   DATA[1580,22] := 1.713645;
   DATA[1580,23] := 795.0654;
   DATA[1580,24] := 2.0;
   DATA[1580,25] := 2.0;
   DATA[1580,26] := 7.876378;
   DATA[1580,27] := 142.8608;
   DATA[1580,28] := 262.8172;
   DATA[1580,29] := 12.11228;
   DATA[1580,30] := 1.724301;
   DATA[1580,31] := 1.291789;
   DATA[1580,32] := 0.7391096;
   DATA[1580,33] := 0.3081703;
   DATA[1580,34] := 2.0;
   DATA[1580,35] := 250.4166;
   DATA[1580,36] := 1.665972;
   DATA[1580,37] := 189.1182;
   DATA[1580,38] := 0.000128152;
   DATA[1580,39] := 1.0;
   DATA[1581,1] := 813.9059;
   DATA[1581,2] := 1.0;
   DATA[1581,3] := 1.0;
   DATA[1581,4] := 262.4968;
   DATA[1581,5] := 8.464369;
   DATA[1581,6] := 319.3027;
   DATA[1581,8] := 1.0;
   DATA[1581,9] := 1.0;
   DATA[1581,10] := 1.0;
   DATA[1581,11] := 19.70677;
   DATA[1581,12] := 2.214265;
   DATA[1581,13] := 907.7801;
   DATA[1581,14] := 1.0;
   DATA[1581,15] := 2.0;
   DATA[1581,16] := 1.0;
   DATA[1581,17] := 1.0;
   DATA[1581,18] := 1.0;
   DATA[1581,19] := 2.0;
   DATA[1581,20] := 148.808;
   DATA[1581,21] := 153.858;
   DATA[1581,22] := 1.713645;
   DATA[1581,23] := 795.2961;
   DATA[1581,24] := 2.0;
   DATA[1581,25] := 2.0;
   DATA[1581,26] := 7.876378;
   DATA[1581,27] := 142.8608;
   DATA[1581,28] := 262.8172;
   DATA[1581,29] := 12.11228;
   DATA[1581,30] := 1.725711;
   DATA[1581,31] := 1.291149;
   DATA[1581,32] := 0.736421;
   DATA[1581,33] := 0.3081703;
   DATA[1581,34] := 2.0;
   DATA[1581,35] := 250.4166;
   DATA[1581,36] := 1.665972;
   DATA[1581,37] := 189.2143;
   DATA[1581,38] := 0.000128152;
   DATA[1581,39] := 1.0;
   DATA[1582,1] := 813.7882;
   DATA[1582,2] := 1.0;
   DATA[1582,3] := 1.0;
   DATA[1582,4] := 262.4968;
   DATA[1582,5] := 8.464369;
   DATA[1582,6] := 319.2771;
   DATA[1582,8] := 1.0;
   DATA[1582,9] := 1.0;
   DATA[1582,10] := 1.0;
   DATA[1582,11] := 19.70677;
   DATA[1582,12] := 2.214265;
   DATA[1582,13] := 907.6199;
   DATA[1582,14] := 1.0;
   DATA[1582,15] := 2.0;
   DATA[1582,16] := 1.0;
   DATA[1582,17] := 1.0;
   DATA[1582,18] := 1.0;
   DATA[1582,19] := 2.0;
   DATA[1582,20] := 148.808;
   DATA[1582,21] := 153.858;
   DATA[1582,22] := 1.713645;
   DATA[1582,23] := 795.3345;
   DATA[1582,24] := 2.0;
   DATA[1582,25] := 2.0;
   DATA[1582,26] := 7.876378;
   DATA[1582,27] := 143.1684;
   DATA[1582,28] := 262.8172;
   DATA[1582,29] := 12.11228;
   DATA[1582,30] := 1.726609;
   DATA[1582,31] := 1.282439;
   DATA[1582,32] := 0.7346286;
   DATA[1582,33] := 0.306761;
   DATA[1582,34] := 2.0;
   DATA[1582,35] := 250.4166;
   DATA[1582,36] := 1.665972;
   DATA[1582,37] := 189.2143;
   DATA[1582,38] := 0.000128152;
   DATA[1582,39] := 1.0;
   DATA[1583,1] := 813.9059;
   DATA[1583,2] := 1.0;
   DATA[1583,3] := 1.0;
   DATA[1583,4] := 262.4968;
   DATA[1583,5] := 8.465651;
   DATA[1583,6] := 319.2258;
   DATA[1583,8] := 1.0;
   DATA[1583,9] := 1.0;
   DATA[1583,10] := 1.0;
   DATA[1583,11] := 19.70677;
   DATA[1583,12] := 2.214265;
   DATA[1583,13] := 906.8989;
   DATA[1583,14] := 1.0;
   DATA[1583,15] := 2.0;
   DATA[1583,16] := 1.0;
   DATA[1583,17] := 1.0;
   DATA[1583,18] := 1.0;
   DATA[1583,19] := 2.0;
   DATA[1583,20] := 148.808;
   DATA[1583,21] := 153.858;
   DATA[1583,22] := 1.715952;
   DATA[1583,23] := 795.7575;
   DATA[1583,24] := 2.0;
   DATA[1583,25] := 2.0;
   DATA[1583,26] := 7.876378;
   DATA[1583,27] := 143.1684;
   DATA[1583,28] := 262.8172;
   DATA[1583,29] := 12.11228;
   DATA[1583,30] := 1.726609;
   DATA[1583,31] := 1.269502;
   DATA[1583,32] := 0.7346286;
   DATA[1583,33] := 0.306761;
   DATA[1583,34] := 2.0;
   DATA[1583,35] := 250.4166;
   DATA[1583,36] := 1.665972;
   DATA[1583,37] := 189.2143;
   DATA[1583,38] := 0.000128152;
   DATA[1583,39] := 1.0;
   DATA[1584,1] := 813.6312;
   DATA[1584,2] := 1.0;
   DATA[1584,3] := 1.0;
   DATA[1584,4] := 262.4968;
   DATA[1584,5] := 8.465651;
   DATA[1584,6] := 319.072;
   DATA[1584,8] := 1.0;
   DATA[1584,9] := 1.0;
   DATA[1584,10] := 1.0;
   DATA[1584,11] := 19.67155;
   DATA[1584,12] := 2.214265;
   DATA[1584,13] := 906.4583;
   DATA[1584,14] := 1.0;
   DATA[1584,15] := 2.0;
   DATA[1584,16] := 1.0;
   DATA[1584,17] := 1.0;
   DATA[1584,18] := 1.0;
   DATA[1584,19] := 2.0;
   DATA[1584,20] := 148.808;
   DATA[1584,21] := 153.858;
   DATA[1584,22] := 1.715952;
   DATA[1584,23] := 795.6806;
   DATA[1584,24] := 2.0;
   DATA[1584,25] := 2.0;
   DATA[1584,26] := 7.876378;
   DATA[1584,27] := 143.1684;
   DATA[1584,28] := 262.8172;
   DATA[1584,29] := 12.11228;
   DATA[1584,30] := 1.726609;
   DATA[1584,31] := 1.261304;
   DATA[1584,32] := 0.7346286;
   DATA[1584,33] := 0.306761;
   DATA[1584,34] := 2.0;
   DATA[1584,35] := 250.4166;
   DATA[1584,36] := 1.665972;
   DATA[1584,37] := 189.2143;
   DATA[1584,38] := 0.000128152;
   DATA[1584,39] := 1.0;
   DATA[1585,1] := 813.5919;
   DATA[1585,2] := 1.0;
   DATA[1585,3] := 1.0;
   DATA[1585,4] := 262.6891;
   DATA[1585,5] := 8.465651;
   DATA[1585,6] := 319.072;
   DATA[1585,8] := 1.0;
   DATA[1585,9] := 1.0;
   DATA[1585,10] := 1.0;
   DATA[1585,11] := 19.67155;
   DATA[1585,12] := 2.214265;
   DATA[1585,13] := 905.6172;
   DATA[1585,14] := 1.0;
   DATA[1585,15] := 2.0;
   DATA[1585,16] := 1.0;
   DATA[1585,17] := 1.0;
   DATA[1585,18] := 1.0;
   DATA[1585,19] := 2.0;
   DATA[1585,20] := 148.808;
   DATA[1585,21] := 153.858;
   DATA[1585,22] := 1.713389;
   DATA[1585,23] := 795.796;
   DATA[1585,24] := 2.0;
   DATA[1585,25] := 2.0;
   DATA[1585,26] := 7.876378;
   DATA[1585,27] := 143.1684;
   DATA[1585,28] := 262.8172;
   DATA[1585,29] := 12.11228;
   DATA[1585,30] := 1.726609;
   DATA[1585,31] := 1.26361;
   DATA[1585,32] := 0.7346286;
   DATA[1585,33] := 0.3084265;
   DATA[1585,34] := 2.0;
   DATA[1585,35] := 250.4166;
   DATA[1585,36] := 1.665972;
   DATA[1585,37] := 189.2143;
   DATA[1585,38] := 0.000128152;
   DATA[1585,39] := 1.0;
   DATA[1586,1] := 813.3956;
   DATA[1586,2] := 1.0;
   DATA[1586,3] := 1.0;
   DATA[1586,4] := 262.6891;
   DATA[1586,5] := 8.465651;
   DATA[1586,6] := 319.072;
   DATA[1586,8] := 1.0;
   DATA[1586,9] := 1.0;
   DATA[1586,10] := 1.0;
   DATA[1586,11] := 19.67155;
   DATA[1586,12] := 2.212856;
   DATA[1586,13] := 905.7774;
   DATA[1586,14] := 1.0;
   DATA[1586,15] := 2.0;
   DATA[1586,16] := 1.0;
   DATA[1586,17] := 1.0;
   DATA[1586,18] := 1.0;
   DATA[1586,19] := 2.0;
   DATA[1586,20] := 148.808;
   DATA[1586,21] := 153.858;
   DATA[1586,22] := 1.713004;
   DATA[1586,23] := 795.796;
   DATA[1586,24] := 2.0;
   DATA[1586,25] := 2.0;
   DATA[1586,26] := 7.874776;
   DATA[1586,27] := 143.0659;
   DATA[1586,28] := 262.8172;
   DATA[1586,29] := 12.11228;
   DATA[1586,30] := 1.726865;
   DATA[1586,31] := 1.271039;
   DATA[1586,32] := 0.7357808;
   DATA[1586,33] := 0.3084265;
   DATA[1586,34] := 2.0;
   DATA[1586,35] := 250.4166;
   DATA[1586,36] := 1.665972;
   DATA[1586,37] := 189.2143;
   DATA[1586,38] := 0.000128152;
   DATA[1586,39] := 1.0;
   DATA[1587,1] := 814.0237;
   DATA[1587,2] := 1.0;
   DATA[1587,3] := 1.0;
   DATA[1587,4] := 262.6891;
   DATA[1587,5] := 8.465651;
   DATA[1587,6] := 319.072;
   DATA[1587,8] := 1.0;
   DATA[1587,9] := 1.0;
   DATA[1587,10] := 1.0;
   DATA[1587,11] := 19.71637;
   DATA[1587,12] := 2.2126;
   DATA[1587,13] := 904.9763;
   DATA[1587,14] := 1.0;
   DATA[1587,15] := 2.0;
   DATA[1587,16] := 1.0;
   DATA[1587,17] := 1.0;
   DATA[1587,18] := 1.0;
   DATA[1587,19] := 2.0;
   DATA[1587,20] := 148.808;
   DATA[1587,21] := 153.9862;
   DATA[1587,22] := 1.713004;
   DATA[1587,23] := 796.1036;
   DATA[1587,24] := 2.0;
   DATA[1587,25] := 2.0;
   DATA[1587,26] := 7.874776;
   DATA[1587,27] := 143.0659;
   DATA[1587,28] := 262.8172;
   DATA[1587,29] := 12.11228;
   DATA[1587,30] := 1.726865;
   DATA[1587,31] := 1.280902;
   DATA[1587,32] := 0.7357808;
   DATA[1587,33] := 0.3084265;
   DATA[1587,34] := 2.0;
   DATA[1587,35] := 250.4166;
   DATA[1587,36] := 1.665972;
   DATA[1587,37] := 189.2143;
   DATA[1587,38] := 0.000128152;
   DATA[1587,39] := 1.0;
   DATA[1588,1] := 813.9844;
   DATA[1588,2] := 1.0;
   DATA[1588,3] := 1.0;
   DATA[1588,4] := 262.6891;
   DATA[1588,5] := 8.465651;
   DATA[1588,6] := 319.072;
   DATA[1588,8] := 1.0;
   DATA[1588,9] := 1.0;
   DATA[1588,10] := 1.0;
   DATA[1588,11] := 19.71637;
   DATA[1588,12] := 2.2126;
   DATA[1588,13] := 904.4957;
   DATA[1588,14] := 1.0;
   DATA[1588,15] := 2.0;
   DATA[1588,16] := 1.0;
   DATA[1588,17] := 1.0;
   DATA[1588,18] := 1.0;
   DATA[1588,19] := 2.0;
   DATA[1588,20] := 148.808;
   DATA[1588,21] := 153.9862;
   DATA[1588,22] := 1.713004;
   DATA[1588,23] := 796.1805;
   DATA[1588,24] := 2.0;
   DATA[1588,25] := 2.0;
   DATA[1588,26] := 7.874776;
   DATA[1588,27] := 143.0659;
   DATA[1588,28] := 262.8172;
   DATA[1588,29] := 12.11228;
   DATA[1588,30] := 1.726865;
   DATA[1588,31] := 1.28167;
   DATA[1588,32] := 0.7357808;
   DATA[1588,33] := 0.3084265;
   DATA[1588,34] := 2.0;
   DATA[1588,35] := 250.4166;
   DATA[1588,36] := 1.665972;
   DATA[1588,37] := 189.2143;
   DATA[1588,38] := 0.000128152;
   DATA[1588,39] := 1.0;
   DATA[1589,1] := 813.7489;
   DATA[1589,2] := 1.0;
   DATA[1589,3] := 1.0;
   DATA[1589,4] := 262.6891;
   DATA[1589,5] := 8.465651;
   DATA[1589,6] := 319.072;
   DATA[1589,8] := 1.0;
   DATA[1589,9] := 1.0;
   DATA[1589,10] := 1.0;
   DATA[1589,11] := 19.74838;
   DATA[1589,12] := 2.2126;
   DATA[1589,13] := 903.8948;
   DATA[1589,14] := 1.0;
   DATA[1589,15] := 2.0;
   DATA[1589,16] := 1.0;
   DATA[1589,17] := 1.0;
   DATA[1589,18] := 1.0;
   DATA[1589,19] := 2.0;
   DATA[1589,20] := 148.808;
   DATA[1589,21] := 153.9862;
   DATA[1589,22] := 1.71262;
   DATA[1589,23] := 795.9498;
   DATA[1589,24] := 2.0;
   DATA[1589,25] := 2.0;
   DATA[1589,26] := 7.874776;
   DATA[1589,27] := 143.0659;
   DATA[1589,28] := 262.8172;
   DATA[1589,29] := 12.11228;
   DATA[1589,30] := 1.726865;
   DATA[1589,31] := 1.279877;
   DATA[1589,32] := 0.7357808;
   DATA[1589,33] := 0.3084265;
   DATA[1589,34] := 2.0;
   DATA[1589,35] := 250.4166;
   DATA[1589,36] := 1.665972;
   DATA[1589,37] := 189.2143;
   DATA[1589,38] := 0.000128152;
   DATA[1589,39] := 1.0;
   DATA[1590,1] := 813.7489;
   DATA[1590,2] := 1.0;
   DATA[1590,3] := 1.0;
   DATA[1590,4] := 262.6891;
   DATA[1590,5] := 8.465651;
   DATA[1590,6] := 319.072;
   DATA[1590,8] := 1.0;
   DATA[1590,9] := 1.0;
   DATA[1590,10] := 1.0;
   DATA[1590,11] := 19.77079;
   DATA[1590,12] := 2.2126;
   DATA[1590,13] := 903.2941;
   DATA[1590,14] := 1.0;
   DATA[1590,15] := 2.0;
   DATA[1590,16] := 1.0;
   DATA[1590,17] := 1.0;
   DATA[1590,18] := 1.0;
   DATA[1590,19] := 2.0;
   DATA[1590,20] := 148.808;
   DATA[1590,21] := 153.9862;
   DATA[1590,22] := 1.711595;
   DATA[1590,23] := 796.3727;
   DATA[1590,24] := 2.0;
   DATA[1590,25] := 2.0;
   DATA[1590,26] := 7.874776;
   DATA[1590,27] := 143.0403;
   DATA[1590,28] := 262.8172;
   DATA[1590,29] := 11.92002;
   DATA[1590,30] := 1.726865;
   DATA[1590,31] := 1.279237;
   DATA[1590,32] := 0.7357808;
   DATA[1590,33] := 0.3084265;
   DATA[1590,34] := 2.0;
   DATA[1590,35] := 250.4166;
   DATA[1590,36] := 1.665972;
   DATA[1590,37] := 189.2143;
   DATA[1590,38] := 0.000128152;
   DATA[1590,39] := 1.0;
   DATA[1591,1] := 813.8275;
   DATA[1591,2] := 1.0;
   DATA[1591,3] := 1.0;
   DATA[1591,4] := 262.6891;
   DATA[1591,5] := 8.465651;
   DATA[1591,6] := 319.072;
   DATA[1591,8] := 1.0;
   DATA[1591,9] := 1.0;
   DATA[1591,10] := 1.0;
   DATA[1591,11] := 19.7996;
   DATA[1591,12] := 2.2126;
   DATA[1591,13] := 902.6532;
   DATA[1591,14] := 1.0;
   DATA[1591,15] := 2.0;
   DATA[1591,16] := 1.0;
   DATA[1591,17] := 1.0;
   DATA[1591,18] := 1.0;
   DATA[1591,19] := 2.0;
   DATA[1591,20] := 148.808;
   DATA[1591,21] := 153.9862;
   DATA[1591,22] := 1.711082;
   DATA[1591,23] := 796.5266;
   DATA[1591,24] := 2.0;
   DATA[1591,25] := 2.0;
   DATA[1591,26] := 7.874776;
   DATA[1591,27] := 143.0403;
   DATA[1591,28] := 262.8172;
   DATA[1591,29] := 11.92002;
   DATA[1591,30] := 1.726865;
   DATA[1591,31] := 1.28167;
   DATA[1591,32] := 0.7352687;
   DATA[1591,33] := 0.3084265;
   DATA[1591,34] := 2.0;
   DATA[1591,35] := 250.4166;
   DATA[1591,36] := 1.665972;
   DATA[1591,37] := 189.2143;
   DATA[1591,38] := 0.000128152;
   DATA[1591,39] := 1.0;
   DATA[1592,1] := 813.5134;
   DATA[1592,2] := 1.0;
   DATA[1592,3] := 1.0;
   DATA[1592,4] := 262.6891;
   DATA[1592,5] := 8.465651;
   DATA[1592,6] := 319.072;
   DATA[1592,8] := 1.0;
   DATA[1592,9] := 1.0;
   DATA[1592,10] := 1.0;
   DATA[1592,11] := 19.7996;
   DATA[1592,12] := 2.211318;
   DATA[1592,13] := 902.2126;
   DATA[1592,14] := 1.0;
   DATA[1592,15] := 2.0;
   DATA[1592,16] := 1.0;
   DATA[1592,17] := 1.0;
   DATA[1592,18] := 1.0;
   DATA[1592,19] := 2.0;
   DATA[1592,20] := 148.808;
   DATA[1592,21] := 153.9862;
   DATA[1592,22] := 1.7098;
   DATA[1592,23] := 796.4496;
   DATA[1592,24] := 2.0;
   DATA[1592,25] := 2.0;
   DATA[1592,26] := 7.874776;
   DATA[1592,27] := 143.0403;
   DATA[1592,28] := 262.8172;
   DATA[1592,29] := 11.92002;
   DATA[1592,30] := 1.726865;
   DATA[1592,31] := 1.291405;
   DATA[1592,32] := 0.7351407;
   DATA[1592,33] := 0.3084265;
   DATA[1592,34] := 2.0;
   DATA[1592,35] := 250.4166;
   DATA[1592,36] := 1.665972;
   DATA[1592,37] := 189.2143;
   DATA[1592,38] := 0.000128152;
   DATA[1592,39] := 1.0;
   DATA[1593,1] := 813.7489;
   DATA[1593,2] := 1.0;
   DATA[1593,3] := 1.0;
   DATA[1593,4] := 262.6891;
   DATA[1593,5] := 8.465651;
   DATA[1593,6] := 319.072;
   DATA[1593,8] := 1.0;
   DATA[1593,9] := 1.0;
   DATA[1593,10] := 1.0;
   DATA[1593,11] := 19.73878;
   DATA[1593,12] := 2.211318;
   DATA[1593,13] := 901.772;
   DATA[1593,14] := 1.0;
   DATA[1593,15] := 2.0;
   DATA[1593,16] := 1.0;
   DATA[1593,17] := 1.0;
   DATA[1593,18] := 1.0;
   DATA[1593,19] := 2.0;
   DATA[1593,20] := 148.808;
   DATA[1593,21] := 153.9862;
   DATA[1593,22] := 1.7098;
   DATA[1593,23] := 796.565;
   DATA[1593,24] := 2.0;
   DATA[1593,25] := 2.0;
   DATA[1593,26] := 7.874776;
   DATA[1593,27] := 143.0403;
   DATA[1593,28] := 262.8172;
   DATA[1593,29] := 11.92002;
   DATA[1593,30] := 1.726865;
   DATA[1593,31] := 1.285641;
   DATA[1593,32] := 0.7351407;
   DATA[1593,33] := 0.3084265;
   DATA[1593,34] := 2.0;
   DATA[1593,35] := 250.4166;
   DATA[1593,36] := 1.665972;
   DATA[1593,37] := 189.2143;
   DATA[1593,38] := 0.000128152;
   DATA[1593,39] := 1.0;
   DATA[1594,1] := 813.5919;
   DATA[1594,2] := 1.0;
   DATA[1594,3] := 1.0;
   DATA[1594,4] := 262.6891;
   DATA[1594,5] := 8.465651;
   DATA[1594,6] := 319.072;
   DATA[1594,8] := 1.0;
   DATA[1594,9] := 1.0;
   DATA[1594,10] := 1.0;
   DATA[1594,11] := 19.73878;
   DATA[1594,12] := 2.2126;
   DATA[1594,13] := 901.2914;
   DATA[1594,14] := 1.0;
   DATA[1594,15] := 2.0;
   DATA[1594,16] := 1.0;
   DATA[1594,17] := 1.0;
   DATA[1594,18] := 1.0;
   DATA[1594,19] := 2.0;
   DATA[1594,20] := 148.808;
   DATA[1594,21] := 153.9862;
   DATA[1594,22] := 1.7098;
   DATA[1594,23] := 797.1418;
   DATA[1594,24] := 2.0;
   DATA[1594,25] := 2.0;
   DATA[1594,26] := 7.874776;
   DATA[1594,27] := 142.8352;
   DATA[1594,28] := 262.8172;
   DATA[1594,29] := 11.92002;
   DATA[1594,30] := 1.726865;
   DATA[1594,31] := 1.289228;
   DATA[1594,32] := 0.7351407;
   DATA[1594,33] := 0.3084265;
   DATA[1594,34] := 2.0;
   DATA[1594,35] := 250.3044;
   DATA[1594,36] := 1.665972;
   DATA[1594,37] := 189.2143;
   DATA[1594,38] := 0.000128152;
   DATA[1594,39] := 1.0;
   DATA[1595,1] := 813.7882;
   DATA[1595,2] := 1.0;
   DATA[1595,3] := 1.0;
   DATA[1595,4] := 262.6891;
   DATA[1595,5] := 8.465651;
   DATA[1595,6] := 319.072;
   DATA[1595,8] := 1.0;
   DATA[1595,9] := 1.0;
   DATA[1595,10] := 1.0;
   DATA[1595,11] := 19.73878;
   DATA[1595,12] := 2.212856;
   DATA[1595,13] := 900.6906;
   DATA[1595,14] := 1.0;
   DATA[1595,15] := 2.0;
   DATA[1595,16] := 1.0;
   DATA[1595,17] := 1.0;
   DATA[1595,18] := 1.0;
   DATA[1595,19] := 2.0;
   DATA[1595,20] := 148.808;
   DATA[1595,21] := 153.9862;
   DATA[1595,22] := 1.7098;
   DATA[1595,23] := 797.0649;
   DATA[1595,24] := 2.0;
   DATA[1595,25] := 2.0;
   DATA[1595,26] := 7.877339;
   DATA[1595,27] := 142.8352;
   DATA[1595,28] := 262.8172;
   DATA[1595,29] := 11.92002;
   DATA[1595,30] := 1.726865;
   DATA[1595,31] := 1.291789;
   DATA[1595,32] := 0.7351407;
   DATA[1595,33] := 0.3084265;
   DATA[1595,34] := 2.0;
   DATA[1595,35] := 250.2724;
   DATA[1595,36] := 1.665972;
   DATA[1595,37] := 188.8939;
   DATA[1595,38] := 0.000128152;
   DATA[1595,39] := 1.0;
   DATA[1596,1] := 813.7882;
   DATA[1596,2] := 1.0;
   DATA[1596,3] := 1.0;
   DATA[1596,4] := 262.6891;
   DATA[1596,5] := 8.465651;
   DATA[1596,6] := 319.072;
   DATA[1596,8] := 1.0;
   DATA[1596,9] := 1.0;
   DATA[1596,10] := 1.0;
   DATA[1596,11] := 19.73878;
   DATA[1596,12] := 2.212856;
   DATA[1596,13] := 900.2499;
   DATA[1596,14] := 1.0;
   DATA[1596,15] := 2.0;
   DATA[1596,16] := 1.0;
   DATA[1596,17] := 1.0;
   DATA[1596,18] := 1.0;
   DATA[1596,19] := 2.0;
   DATA[1596,20] := 148.808;
   DATA[1596,21] := 153.9862;
   DATA[1596,22] := 1.7098;
   DATA[1596,23] := 797.2187;
   DATA[1596,24] := 2.0;
   DATA[1596,25] := 2.0;
   DATA[1596,26] := 7.877339;
   DATA[1596,27] := 142.8352;
   DATA[1596,28] := 262.8172;
   DATA[1596,29] := 12.26609;
   DATA[1596,30] := 1.725968;
   DATA[1596,31] := 1.291789;
   DATA[1596,32] := 0.7351407;
   DATA[1596,33] := 0.3084265;
   DATA[1596,34] := 2.0;
   DATA[1596,35] := 250.0801;
   DATA[1596,36] := 1.665972;
   DATA[1596,37] := 188.8779;
   DATA[1596,38] := 0.000128152;
   DATA[1596,39] := 1.0;
   DATA[1597,1] := 813.6312;
   DATA[1597,2] := 1.0;
   DATA[1597,3] := 1.0;
   DATA[1597,4] := 262.4648;
   DATA[1597,5] := 8.465651;
   DATA[1597,6] := 319.072;
   DATA[1597,8] := 1.0;
   DATA[1597,9] := 1.0;
   DATA[1597,10] := 1.0;
   DATA[1597,11] := 19.75159;
   DATA[1597,12] := 2.212856;
   DATA[1597,13] := 899.7693;
   DATA[1597,14] := 1.0;
   DATA[1597,15] := 2.0;
   DATA[1597,16] := 1.0;
   DATA[1597,17] := 1.0;
   DATA[1597,18] := 1.0;
   DATA[1597,19] := 2.0;
   DATA[1597,20] := 148.808;
   DATA[1597,21] := 153.9862;
   DATA[1597,22] := 1.7098;
   DATA[1597,23] := 797.4494;
   DATA[1597,24] := 2.0;
   DATA[1597,25] := 2.0;
   DATA[1597,26] := 7.877339;
   DATA[1597,27] := 142.8352;
   DATA[1597,28] := 262.8172;
   DATA[1597,29] := 12.26609;
   DATA[1597,30] := 1.724301;
   DATA[1597,31] := 1.301652;
   DATA[1597,32] := 0.7351407;
   DATA[1597,33] := 0.3084265;
   DATA[1597,34] := 2.0;
   DATA[1597,35] := 250.0801;
   DATA[1597,36] := 1.665972;
   DATA[1597,37] := 188.8779;
   DATA[1597,38] := 0.000128152;
   DATA[1597,39] := 1.0;
   DATA[1598,1] := 813.5134;
   DATA[1598,2] := 1.0;
   DATA[1598,3] := 1.0;
   DATA[1598,4] := 262.4648;
   DATA[1598,5] := 8.466612;
   DATA[1598,6] := 319.072;
   DATA[1598,8] := 1.0;
   DATA[1598,9] := 1.0;
   DATA[1598,10] := 1.0;
   DATA[1598,11] := 19.7804;
   DATA[1598,12] := 2.212856;
   DATA[1598,13] := 899.4489;
   DATA[1598,14] := 1.0;
   DATA[1598,15] := 2.0;
   DATA[1598,16] := 1.0;
   DATA[1598,17] := 1.0;
   DATA[1598,18] := 1.0;
   DATA[1598,19] := 2.0;
   DATA[1598,20] := 148.808;
   DATA[1598,21] := 153.9862;
   DATA[1598,22] := 1.7098;
   DATA[1598,23] := 797.5262;
   DATA[1598,24] := 2.0;
   DATA[1598,25] := 2.0;
   DATA[1598,26] := 7.877339;
   DATA[1598,27] := 143.0403;
   DATA[1598,28] := 262.8172;
   DATA[1598,29] := 12.26609;
   DATA[1598,30] := 1.722379;
   DATA[1598,31] := 1.294095;
   DATA[1598,32] := 0.7351407;
   DATA[1598,33] := 0.3074656;
   DATA[1598,34] := 2.0;
   DATA[1598,35] := 249.9359;
   DATA[1598,36] := 1.665972;
   DATA[1598,37] := 188.8779;
   DATA[1598,38] := 0.000128152;
   DATA[1598,39] := 1.0;
   DATA[1599,1] := 813.9059;
   DATA[1599,2] := 1.0;
   DATA[1599,3] := 1.0;
   DATA[1599,4] := 262.4648;
   DATA[1599,5] := 8.467573;
   DATA[1599,6] := 319.072;
   DATA[1599,8] := 1.0;
   DATA[1599,9] := 1.0;
   DATA[1599,10] := 1.0;
   DATA[1599,11] := 19.7964;
   DATA[1599,12] := 2.212856;
   DATA[1599,13] := 898.9282;
   DATA[1599,14] := 1.0;
   DATA[1599,15] := 2.0;
   DATA[1599,16] := 1.0;
   DATA[1599,17] := 1.0;
   DATA[1599,18] := 1.0;
   DATA[1599,19] := 2.0;
   DATA[1599,20] := 148.808;
   DATA[1599,21] := 153.9093;
   DATA[1599,22] := 1.7098;
   DATA[1599,23] := 797.4879;
   DATA[1599,24] := 2.0;
   DATA[1599,25] := 2.0;
   DATA[1599,26] := 7.877339;
   DATA[1599,27] := 143.0403;
   DATA[1599,28] := 262.8172;
   DATA[1599,29] := 12.26609;
   DATA[1599,30] := 1.722379;
   DATA[1599,31] := 1.291533;
   DATA[1599,32] := 0.7351407;
   DATA[1599,33] := 0.3074656;
   DATA[1599,34] := 2.0;
   DATA[1599,35] := 249.9359;
   DATA[1599,36] := 1.665972;
   DATA[1599,37] := 188.8779;
   DATA[1599,38] := 0.000128152;
   DATA[1599,39] := 1.0;
   DATA[1600,1] := 814.2985;
   DATA[1600,2] := 1.0;
   DATA[1600,3] := 1.0;
   DATA[1600,4] := 262.4648;
   DATA[1600,5] := 8.467573;
   DATA[1600,6] := 319.072;
   DATA[1600,8] := 1.0;
   DATA[1600,9] := 1.0;
   DATA[1600,10] := 1.0;
   DATA[1600,11] := 19.7964;
   DATA[1600,12] := 2.212856;
   DATA[1600,13] := 898.8481;
   DATA[1600,14] := 1.0;
   DATA[1600,15] := 2.0;
   DATA[1600,16] := 1.0;
   DATA[1600,17] := 1.0;
   DATA[1600,18] := 1.0;
   DATA[1600,19] := 2.0;
   DATA[1600,20] := 148.808;
   DATA[1600,21] := 153.858;
   DATA[1600,22] := 1.7098;
   DATA[1600,23] := 797.6416;
   DATA[1600,24] := 2.0;
   DATA[1600,25] := 2.0;
   DATA[1600,26] := 7.877339;
   DATA[1600,27] := 143.0403;
   DATA[1600,28] := 262.8172;
   DATA[1600,29] := 12.07383;
   DATA[1600,30] := 1.720969;
   DATA[1600,31] := 1.291533;
   DATA[1600,32] := 0.7351407;
   DATA[1600,33] := 0.3084265;
   DATA[1600,34] := 2.0;
   DATA[1600,35] := 249.9359;
   DATA[1600,36] := 1.665972;
   DATA[1600,37] := 188.8779;
   DATA[1600,38] := 0.000128152;
   DATA[1600,39] := 1.0;
   DATA[1601,1] := 814.1415;
   DATA[1601,2] := 1.0;
   DATA[1601,3] := 1.0;
   DATA[1601,4] := 262.5609;
   DATA[1601,5] := 8.467573;
   DATA[1601,6] := 319.072;
   DATA[1601,8] := 1.0;
   DATA[1601,9] := 1.0;
   DATA[1601,10] := 1.0;
   DATA[1601,11] := 19.8028;
   DATA[1601,12] := 2.212856;
   DATA[1601,13] := 898.3274;
   DATA[1601,14] := 1.0;
   DATA[1601,15] := 2.0;
   DATA[1601,16] := 1.0;
   DATA[1601,17] := 1.0;
   DATA[1601,18] := 1.0;
   DATA[1601,19] := 2.0;
   DATA[1601,20] := 148.808;
   DATA[1601,21] := 153.858;
   DATA[1601,22] := 1.7098;
   DATA[1601,23] := 797.4494;
   DATA[1601,24] := 2.0;
   DATA[1601,25] := 2.0;
   DATA[1601,26] := 7.877339;
   DATA[1601,27] := 143.0403;
   DATA[1601,28] := 262.4648;
   DATA[1601,29] := 12.07383;
   DATA[1601,30] := 1.720969;
   DATA[1601,31] := 1.291533;
   DATA[1601,32] := 0.7351407;
   DATA[1601,33] := 0.3084265;
   DATA[1601,34] := 2.0;
   DATA[1601,35] := 249.9359;
   DATA[1601,36] := 1.665972;
   DATA[1601,37] := 188.8779;
   DATA[1601,38] := 0.000128152;
   DATA[1601,39] := 1.0;
   DATA[1602,1] := 814.1022;
   DATA[1602,2] := 1.0;
   DATA[1602,3] := 1.0;
   DATA[1602,4] := 262.6891;
   DATA[1602,5] := 8.467573;
   DATA[1602,6] := 319.072;
   DATA[1602,8] := 1.0;
   DATA[1602,9] := 1.0;
   DATA[1602,10] := 1.0;
   DATA[1602,11] := 19.8028;
   DATA[1602,12] := 2.212856;
   DATA[1602,13] := 897.4061;
   DATA[1602,14] := 1.0;
   DATA[1602,15] := 2.0;
   DATA[1602,16] := 1.0;
   DATA[1602,17] := 1.0;
   DATA[1602,18] := 1.0;
   DATA[1602,19] := 2.0;
   DATA[1602,20] := 148.808;
   DATA[1602,21] := 153.858;
   DATA[1602,22] := 1.7098;
   DATA[1602,23] := 797.8723;
   DATA[1602,24] := 2.0;
   DATA[1602,25] := 2.0;
   DATA[1602,26] := 7.877339;
   DATA[1602,27] := 143.0403;
   DATA[1602,28] := 262.4648;
   DATA[1602,29] := 12.07383;
   DATA[1602,30] := 1.720969;
   DATA[1602,31] := 1.291533;
   DATA[1602,32] := 0.7351407;
   DATA[1602,33] := 0.3084265;
   DATA[1602,34] := 2.0;
   DATA[1602,35] := 249.984;
   DATA[1602,36] := 1.665972;
   DATA[1602,37] := 188.8779;
   DATA[1602,38] := 0.000128152;
   DATA[1602,39] := 1.0;
   DATA[1603,1] := 814.1022;
   DATA[1603,2] := 1.0;
   DATA[1603,3] := 1.0;
   DATA[1603,4] := 262.6891;
   DATA[1603,5] := 8.467573;
   DATA[1603,6] := 319.072;
   DATA[1603,8] := 1.0;
   DATA[1603,9] := 1.0;
   DATA[1603,10] := 1.0;
   DATA[1603,11] := 19.8028;
   DATA[1603,12] := 2.212856;
   DATA[1603,13] := 897.1257;
   DATA[1603,14] := 1.0;
   DATA[1603,15] := 2.0;
   DATA[1603,16] := 1.0;
   DATA[1603,17] := 1.0;
   DATA[1603,18] := 1.0;
   DATA[1603,19] := 2.0;
   DATA[1603,20] := 148.808;
   DATA[1603,21] := 153.858;
   DATA[1603,22] := 1.7098;
   DATA[1603,23] := 798.2184;
   DATA[1603,24] := 2.0;
   DATA[1603,25] := 2.0;
   DATA[1603,26] := 7.877339;
   DATA[1603,27] := 143.0403;
   DATA[1603,28] := 262.657;
   DATA[1603,29] := 12.07383;
   DATA[1603,30] := 1.720969;
   DATA[1603,31] := 1.272064;
   DATA[1603,32] := 0.7351407;
   DATA[1603,33] := 0.3084265;
   DATA[1603,34] := 2.0;
   DATA[1603,35] := 250.0801;
   DATA[1603,36] := 1.665972;
   DATA[1603,37] := 188.8779;
   DATA[1603,38] := 0.000128152;
   DATA[1603,39] := 1.0;
   DATA[1604,1] := 814.3377;
   DATA[1604,2] := 1.0;
   DATA[1604,3] := 1.0;
   DATA[1604,4] := 262.6891;
   DATA[1604,5] := 8.467573;
   DATA[1604,6] := 319.072;
   DATA[1604,8] := 1.0;
   DATA[1604,9] := 1.0;
   DATA[1604,10] := 1.0;
   DATA[1604,11] := 19.8028;
   DATA[1604,12] := 2.212856;
   DATA[1604,13] := 896.7252;
   DATA[1604,14] := 1.0;
   DATA[1604,15] := 2.0;
   DATA[1604,16] := 1.0;
   DATA[1604,17] := 1.0;
   DATA[1604,18] := 1.0;
   DATA[1604,19] := 2.0;
   DATA[1604,20] := 148.808;
   DATA[1604,21] := 153.858;
   DATA[1604,22] := 1.7098;
   DATA[1604,23] := 797.7954;
   DATA[1604,24] := 2.0;
   DATA[1604,25] := 2.0;
   DATA[1604,26] := 7.877339;
   DATA[1604,27] := 142.9121;
   DATA[1604,28] := 262.8493;
   DATA[1604,29] := 12.07383;
   DATA[1604,30] := 1.721738;
   DATA[1604,31] := 1.255284;
   DATA[1604,32] := 0.7351407;
   DATA[1604,33] := 0.3084265;
   DATA[1604,34] := 2.0;
   DATA[1604,35] := 250.0801;
   DATA[1604,36] := 1.665972;
   DATA[1604,37] := 188.8779;
   DATA[1604,38] := 0.000128152;
   DATA[1604,39] := 1.0;
   DATA[1605,1] := 814.6125;
   DATA[1605,2] := 1.0;
   DATA[1605,3] := 1.0;
   DATA[1605,4] := 262.6891;
   DATA[1605,5] := 8.470778;
   DATA[1605,6] := 319.072;
   DATA[1605,8] := 1.0;
   DATA[1605,9] := 1.0;
   DATA[1605,10] := 1.0;
   DATA[1605,11] := 19.8028;
   DATA[1605,12] := 2.212856;
   DATA[1605,13] := 896.4448;
   DATA[1605,14] := 1.0;
   DATA[1605,15] := 2.0;
   DATA[1605,16] := 1.0;
   DATA[1605,17] := 1.0;
   DATA[1605,18] := 1.0;
   DATA[1605,19] := 2.0;
   DATA[1605,20] := 148.808;
   DATA[1605,21] := 153.858;
   DATA[1605,22] := 1.711338;
   DATA[1605,23] := 797.8723;
   DATA[1605,24] := 2.0;
   DATA[1605,25] := 2.0;
   DATA[1605,26] := 7.877339;
   DATA[1605,27] := 142.9121;
   DATA[1605,28] := 262.8493;
   DATA[1605,29] := 12.07383;
   DATA[1605,30] := 1.721738;
   DATA[1605,31] := 1.254131;
   DATA[1605,32] := 0.7351407;
   DATA[1605,33] := 0.3098997;
   DATA[1605,34] := 2.0;
   DATA[1605,35] := 250.0801;
   DATA[1605,36] := 1.665972;
   DATA[1605,37] := 188.8779;
   DATA[1605,38] := 0.000128152;
   DATA[1605,39] := 1.0;
   DATA[1606,1] := 814.6125;
   DATA[1606,2] := 1.0;
   DATA[1606,3] := 1.0;
   DATA[1606,4] := 262.6891;
   DATA[1606,5] := 8.470778;
   DATA[1606,6] := 319.072;
   DATA[1606,8] := 1.0;
   DATA[1606,9] := 1.0;
   DATA[1606,10] := 1.0;
   DATA[1606,11] := 19.84442;
   DATA[1606,12] := 2.213881;
   DATA[1606,13] := 895.5637;
   DATA[1606,14] := 1.0;
   DATA[1606,15] := 2.0;
   DATA[1606,16] := 1.0;
   DATA[1606,17] := 1.0;
   DATA[1606,18] := 1.0;
   DATA[1606,19] := 2.0;
   DATA[1606,20] := 148.808;
   DATA[1606,21] := 153.858;
   DATA[1606,22] := 1.711979;
   DATA[1606,23] := 798.2184;
   DATA[1606,24] := 2.0;
   DATA[1606,25] := 2.0;
   DATA[1606,26] := 7.877339;
   DATA[1606,27] := 142.9121;
   DATA[1606,28] := 262.8493;
   DATA[1606,29] := 12.07383;
   DATA[1606,30] := 1.721738;
   DATA[1606,31] := 1.253619;
   DATA[1606,32] := 0.7351407;
   DATA[1606,33] := 0.3104122;
   DATA[1606,34] := 2.0;
   DATA[1606,35] := 250.0641;
   DATA[1606,36] := 1.665972;
   DATA[1606,37] := 188.8779;
   DATA[1606,38] := 0.000128152;
   DATA[1606,39] := 1.0;
   DATA[1607,1] := 814.5732;
   DATA[1607,2] := 1.0;
   DATA[1607,3] := 1.0;
   DATA[1607,4] := 262.5288;
   DATA[1607,5] := 8.470778;
   DATA[1607,6] := 319.072;
   DATA[1607,8] := 1.0;
   DATA[1607,9] := 1.0;
   DATA[1607,10] := 1.0;
   DATA[1607,11] := 19.84442;
   DATA[1607,12] := 2.213881;
   DATA[1607,13] := 894.8427;
   DATA[1607,14] := 1.0;
   DATA[1607,15] := 2.0;
   DATA[1607,16] := 1.0;
   DATA[1607,17] := 1.0;
   DATA[1607,18] := 1.0;
   DATA[1607,19] := 2.0;
   DATA[1607,20] := 148.808;
   DATA[1607,21] := 154.0631;
   DATA[1607,22] := 1.711979;
   DATA[1607,23] := 797.6416;
   DATA[1607,24] := 2.0;
   DATA[1607,25] := 2.0;
   DATA[1607,26] := 7.877339;
   DATA[1607,27] := 142.9121;
   DATA[1607,28] := 262.8493;
   DATA[1607,29] := 12.07383;
   DATA[1607,30] := 1.721738;
   DATA[1607,31] := 1.268477;
   DATA[1607,32] := 0.7351407;
   DATA[1607,33] := 0.309003;
   DATA[1607,34] := 2.0;
   DATA[1607,35] := 249.9359;
   DATA[1607,36] := 1.665972;
   DATA[1607,37] := 188.8779;
   DATA[1607,38] := 0.000128152;
   DATA[1607,39] := 1.0;
   DATA[1608,1] := 814.7302;
   DATA[1608,2] := 1.0;
   DATA[1608,3] := 1.0;
   DATA[1608,4] := 262.5288;
   DATA[1608,5] := 8.470778;
   DATA[1608,6] := 319.072;
   DATA[1608,8] := 1.0;
   DATA[1608,9] := 1.0;
   DATA[1608,10] := 1.0;
   DATA[1608,11] := 19.81241;
   DATA[1608,12] := 2.213881;
   DATA[1608,13] := 894.9228;
   DATA[1608,14] := 1.0;
   DATA[1608,15] := 2.0;
   DATA[1608,16] := 1.0;
   DATA[1608,17] := 1.0;
   DATA[1608,18] := 1.0;
   DATA[1608,19] := 2.0;
   DATA[1608,20] := 148.808;
   DATA[1608,21] := 154.0631;
   DATA[1608,22] := 1.713517;
   DATA[1608,23] := 797.6031;
   DATA[1608,24] := 2.0;
   DATA[1608,25] := 2.0;
   DATA[1608,26] := 7.875737;
   DATA[1608,27] := 142.9121;
   DATA[1608,28] := 262.8493;
   DATA[1608,29] := 12.07383;
   DATA[1608,30] := 1.721738;
   DATA[1608,31] := 1.286666;
   DATA[1608,32] := 0.7351407;
   DATA[1608,33] := 0.309003;
   DATA[1608,34] := 2.0;
   DATA[1608,35] := 249.9359;
   DATA[1608,36] := 1.665972;
   DATA[1608,37] := 188.8779;
   DATA[1608,38] := 0.000128152;
   DATA[1608,39] := 1.0;
   DATA[1609,1] := 814.7695;
   DATA[1609,2] := 1.0;
   DATA[1609,3] := 1.0;
   DATA[1609,4] := 262.5288;
   DATA[1609,5] := 8.468214;
   DATA[1609,6] := 319.072;
   DATA[1609,8] := 1.0;
   DATA[1609,9] := 1.0;
   DATA[1609,10] := 1.0;
   DATA[1609,11] := 19.7996;
   DATA[1609,12] := 2.211447;
   DATA[1609,13] := 894.2419;
   DATA[1609,14] := 1.0;
   DATA[1609,15] := 2.0;
   DATA[1609,16] := 1.0;
   DATA[1609,17] := 1.0;
   DATA[1609,18] := 1.0;
   DATA[1609,19] := 2.0;
   DATA[1609,20] := 148.808;
   DATA[1609,21] := 154.0631;
   DATA[1609,22] := 1.713517;
   DATA[1609,23] := 797.8339;
   DATA[1609,24] := 2.0;
   DATA[1609,25] := 2.0;
   DATA[1609,26] := 7.875737;
   DATA[1609,27] := 142.9121;
   DATA[1609,28] := 262.8493;
   DATA[1609,29] := 12.07383;
   DATA[1609,30] := 1.721738;
   DATA[1609,31] := 1.283848;
   DATA[1609,32] := 0.7351407;
   DATA[1609,33] := 0.309003;
   DATA[1609,34] := 2.0;
   DATA[1609,35] := 249.9359;
   DATA[1609,36] := 1.665972;
   DATA[1609,37] := 188.8779;
   DATA[1609,38] := 0.000128152;
   DATA[1609,39] := 1.0;
   DATA[1610,1] := 814.4948;
   DATA[1610,2] := 1.0;
   DATA[1610,3] := 1.0;
   DATA[1610,4] := 262.5288;
   DATA[1610,5] := 8.468214;
   DATA[1610,6] := 319.072;
   DATA[1610,8] := 1.0;
   DATA[1610,9] := 1.0;
   DATA[1610,10] := 1.0;
   DATA[1610,11] := 19.7996;
   DATA[1610,12] := 2.211447;
   DATA[1610,13] := 894.1618;
   DATA[1610,14] := 1.0;
   DATA[1610,15] := 2.0;
   DATA[1610,16] := 1.0;
   DATA[1610,17] := 1.0;
   DATA[1610,18] := 1.0;
   DATA[1610,19] := 2.0;
   DATA[1610,20] := 148.808;
   DATA[1610,21] := 154.0631;
   DATA[1610,22] := 1.712363;
   DATA[1610,23] := 797.6801;
   DATA[1610,24] := 2.0;
   DATA[1610,25] := 2.0;
   DATA[1610,26] := 7.875737;
   DATA[1610,27] := 142.9121;
   DATA[1610,28] := 262.8493;
   DATA[1610,29] := 12.07383;
   DATA[1610,30] := 1.721738;
   DATA[1610,31] := 1.27834;
   DATA[1610,32] := 0.7351407;
   DATA[1610,33] := 0.3083624;
   DATA[1610,34] := 2.0;
   DATA[1610,35] := 249.9359;
   DATA[1610,36] := 1.665972;
   DATA[1610,37] := 188.8779;
   DATA[1610,38] := 0.000128152;
   DATA[1610,39] := 1.0;
   DATA[1611,1] := 814.4948;
   DATA[1611,2] := 1.0;
   DATA[1611,3] := 1.0;
   DATA[1611,4] := 262.5288;
   DATA[1611,5] := 8.468214;
   DATA[1611,6] := 319.072;
   DATA[1611,8] := 1.0;
   DATA[1611,9] := 1.0;
   DATA[1611,10] := 1.0;
   DATA[1611,11] := 19.7996;
   DATA[1611,12] := 2.211447;
   DATA[1611,13] := 893.4408;
   DATA[1611,14] := 1.0;
   DATA[1611,15] := 2.0;
   DATA[1611,16] := 1.0;
   DATA[1611,17] := 1.0;
   DATA[1611,18] := 1.0;
   DATA[1611,19] := 2.0;
   DATA[1611,20] := 148.808;
   DATA[1611,21] := 154.0631;
   DATA[1611,22] := 1.711723;
   DATA[1611,23] := 797.7185;
   DATA[1611,24] := 2.0;
   DATA[1611,25] := 2.0;
   DATA[1611,26] := 7.875737;
   DATA[1611,27] := 142.9121;
   DATA[1611,28] := 262.8493;
   DATA[1611,29] := 12.07383;
   DATA[1611,30] := 1.721738;
   DATA[1611,31] := 1.269374;
   DATA[1611,32] := 0.7351407;
   DATA[1611,33] := 0.3082983;
   DATA[1611,34] := 2.0;
   DATA[1611,35] := 249.9359;
   DATA[1611,36] := 1.665972;
   DATA[1611,37] := 188.8779;
   DATA[1611,38] := 0.000128152;
   DATA[1611,39] := 1.0;
   DATA[1612,1] := 815.005;
   DATA[1612,2] := 1.0;
   DATA[1612,3] := 1.0;
   DATA[1612,4] := 262.5288;
   DATA[1612,5] := 8.468214;
   DATA[1612,6] := 319.072;
   DATA[1612,8] := 1.0;
   DATA[1612,9] := 1.0;
   DATA[1612,10] := 1.0;
   DATA[1612,11] := 19.7996;
   DATA[1612,12] := 2.212343;
   DATA[1612,13] := 893.4008;
   DATA[1612,14] := 1.0;
   DATA[1612,15] := 2.0;
   DATA[1612,16] := 1.0;
   DATA[1612,17] := 1.0;
   DATA[1612,18] := 1.0;
   DATA[1612,19] := 2.0;
   DATA[1612,20] := 148.808;
   DATA[1612,21] := 154.0631;
   DATA[1612,22] := 1.711723;
   DATA[1612,23] := 797.8723;
   DATA[1612,24] := 2.0;
   DATA[1612,25] := 2.0;
   DATA[1612,26] := 7.875737;
   DATA[1612,27] := 142.9121;
   DATA[1612,28] := 262.8172;
   DATA[1612,29] := 12.07383;
   DATA[1612,30] := 1.721738;
   DATA[1612,31] := 1.261432;
   DATA[1612,32] := 0.7351407;
   DATA[1612,33] := 0.3082983;
   DATA[1612,34] := 2.0;
   DATA[1612,35] := 250.1923;
   DATA[1612,36] := 1.665972;
   DATA[1612,37] := 188.8779;
   DATA[1612,38] := 0.000128152;
   DATA[1612,39] := 1.0;
   DATA[1613,1] := 814.9658;
   DATA[1613,2] := 1.0;
   DATA[1613,3] := 1.0;
   DATA[1613,4] := 262.5288;
   DATA[1613,5] := 8.468214;
   DATA[1613,6] := 319.0977;
   DATA[1613,8] := 1.0;
   DATA[1613,9] := 1.0;
   DATA[1613,10] := 1.0;
   DATA[1613,11] := 19.80601;
   DATA[1613,12] := 2.213496;
   DATA[1613,13] := 892.7599;
   DATA[1613,14] := 1.0;
   DATA[1613,15] := 2.0;
   DATA[1613,16] := 1.0;
   DATA[1613,17] := 1.0;
   DATA[1613,18] := 1.0;
   DATA[1613,19] := 2.0;
   DATA[1613,20] := 148.808;
   DATA[1613,21] := 154.0631;
   DATA[1613,22] := 1.711723;
   DATA[1613,23] := 797.7185;
   DATA[1613,24] := 2.0;
   DATA[1613,25] := 2.0;
   DATA[1613,26] := 7.875737;
   DATA[1613,27] := 142.9121;
   DATA[1613,28] := 262.8172;
   DATA[1613,29] := 12.07383;
   DATA[1613,30] := 1.721738;
   DATA[1613,31] := 1.268093;
   DATA[1613,32] := 0.7351407;
   DATA[1613,33] := 0.3082983;
   DATA[1613,34] := 2.0;
   DATA[1613,35] := 250.1923;
   DATA[1613,36] := 1.665972;
   DATA[1613,37] := 188.8779;
   DATA[1613,38] := 0.000128152;
   DATA[1613,39] := 1.0;
   DATA[1614,1] := 815.005;
   DATA[1614,2] := 1.0;
   DATA[1614,3] := 1.0;
   DATA[1614,4] := 262.5288;
   DATA[1614,5] := 8.468214;
   DATA[1614,6] := 319.1489;
   DATA[1614,8] := 1.0;
   DATA[1614,9] := 1.0;
   DATA[1614,10] := 1.0;
   DATA[1614,11] := 19.80601;
   DATA[1614,12] := 2.213496;
   DATA[1614,13] := 892.1992;
   DATA[1614,14] := 1.0;
   DATA[1614,15] := 2.0;
   DATA[1614,16] := 1.0;
   DATA[1614,17] := 1.0;
   DATA[1614,18] := 1.0;
   DATA[1614,19] := 2.0;
   DATA[1614,20] := 148.808;
   DATA[1614,21] := 154.0631;
   DATA[1614,22] := 1.711723;
   DATA[1614,23] := 797.7954;
   DATA[1614,24] := 2.0;
   DATA[1614,25] := 2.0;
   DATA[1614,26] := 7.875737;
   DATA[1614,27] := 142.9121;
   DATA[1614,28] := 262.8172;
   DATA[1614,29] := 12.07383;
   DATA[1614,30] := 1.721738;
   DATA[1614,31] := 1.272064;
   DATA[1614,32] := 0.7351407;
   DATA[1614,33] := 0.3082983;
   DATA[1614,34] := 2.0;
   DATA[1614,35] := 250.1762;
   DATA[1614,36] := 1.665972;
   DATA[1614,37] := 188.8779;
   DATA[1614,38] := 0.000128152;
   DATA[1614,39] := 1.0;
   DATA[1615,1] := 814.9265;
   DATA[1615,2] := 1.0;
   DATA[1615,3] := 1.0;
   DATA[1615,4] := 262.5288;
   DATA[1615,5] := 8.468214;
   DATA[1615,6] := 319.1746;
   DATA[1615,8] := 1.0;
   DATA[1615,9] := 1.0;
   DATA[1615,10] := 1.0;
   DATA[1615,11] := 19.7804;
   DATA[1615,12] := 2.213496;
   DATA[1615,13] := 891.8386;
   DATA[1615,14] := 1.0;
   DATA[1615,15] := 2.0;
   DATA[1615,16] := 1.0;
   DATA[1615,17] := 1.0;
   DATA[1615,18] := 1.0;
   DATA[1615,19] := 2.0;
   DATA[1615,20] := 148.808;
   DATA[1615,21] := 154.0631;
   DATA[1615,22] := 1.71262;
   DATA[1615,23] := 798.1799;
   DATA[1615,24] := 2.0;
   DATA[1615,25] := 2.0;
   DATA[1615,26] := 7.875737;
   DATA[1615,27] := 142.9121;
   DATA[1615,28] := 262.7852;
   DATA[1615,29] := 12.07383;
   DATA[1615,30] := 1.72302;
   DATA[1615,31] := 1.272064;
   DATA[1615,32] := 0.7351407;
   DATA[1615,33] := 0.3082983;
   DATA[1615,34] := 2.0;
   DATA[1615,35] := 250.016;
   DATA[1615,36] := 1.665972;
   DATA[1615,37] := 188.8779;
   DATA[1615,38] := 0.000128152;
   DATA[1615,39] := 1.0;
   DATA[1616,1] := 815.2013;
   DATA[1616,2] := 1.0;
   DATA[1616,3] := 1.0;
   DATA[1616,4] := 262.6891;
   DATA[1616,5] := 8.468214;
   DATA[1616,6] := 319.2771;
   DATA[1616,8] := 1.0;
   DATA[1616,9] := 1.0;
   DATA[1616,10] := 1.0;
   DATA[1616,11] := 19.68436;
   DATA[1616,12] := 2.2126;
   DATA[1616,13] := 891.358;
   DATA[1616,14] := 1.0;
   DATA[1616,15] := 2.0;
   DATA[1616,16] := 1.0;
   DATA[1616,17] := 1.0;
   DATA[1616,18] := 1.0;
   DATA[1616,19] := 2.0;
   DATA[1616,20] := 148.808;
   DATA[1616,21] := 154.0631;
   DATA[1616,22] := 1.71262;
   DATA[1616,23] := 798.4106;
   DATA[1616,24] := 2.0;
   DATA[1616,25] := 2.0;
   DATA[1616,26] := 7.875737;
   DATA[1616,27] := 142.9121;
   DATA[1616,28] := 262.657;
   DATA[1616,29] := 12.07383;
   DATA[1616,30] := 1.723789;
   DATA[1616,31] := 1.272704;
   DATA[1616,32] := 0.7351407;
   DATA[1616,33] := 0.3082983;
   DATA[1616,34] := 2.0;
   DATA[1616,35] := 250.016;
   DATA[1616,36] := 1.665972;
   DATA[1616,37] := 188.8779;
   DATA[1616,38] := 0.000128152;
   DATA[1616,39] := 1.0;
   DATA[1617,1] := 815.005;
   DATA[1617,2] := 1.0;
   DATA[1617,3] := 1.0;
   DATA[1617,4] := 262.7211;
   DATA[1617,5] := 8.468214;
   DATA[1617,6] := 319.2771;
   DATA[1617,8] := 1.0;
   DATA[1617,9] := 1.0;
   DATA[1617,10] := 1.0;
   DATA[1617,11] := 19.66835;
   DATA[1617,12] := 2.2126;
   DATA[1617,13] := 891.0376;
   DATA[1617,14] := 1.0;
   DATA[1617,15] := 2.0;
   DATA[1617,16] := 1.0;
   DATA[1617,17] := 1.0;
   DATA[1617,18] := 1.0;
   DATA[1617,19] := 2.0;
   DATA[1617,20] := 148.808;
   DATA[1617,21] := 154.0631;
   DATA[1617,22] := 1.71262;
   DATA[1617,23] := 798.4106;
   DATA[1617,24] := 2.0;
   DATA[1617,25] := 2.0;
   DATA[1617,26] := 7.875737;
   DATA[1617,27] := 142.6045;
   DATA[1617,28] := 262.657;
   DATA[1617,29] := 12.07383;
   DATA[1617,30] := 1.723789;
   DATA[1617,31] := 1.280646;
   DATA[1617,32] := 0.7351407;
   DATA[1617,33] := 0.3082983;
   DATA[1617,34] := 2.0;
   DATA[1617,35] := 250.016;
   DATA[1617,36] := 1.665972;
   DATA[1617,37] := 188.8779;
   DATA[1617,38] := 0.000128152;
   DATA[1617,39] := 1.0;
   DATA[1618,1] := 815.005;
   DATA[1618,2] := 1.0;
   DATA[1618,3] := 1.0;
   DATA[1618,4] := 262.7211;
   DATA[1618,5] := 8.466612;
   DATA[1618,6] := 319.2771;
   DATA[1618,8] := 1.0;
   DATA[1618,9] := 1.0;
   DATA[1618,10] := 1.0;
   DATA[1618,11] := 19.70037;
   DATA[1618,12] := 2.213881;
   DATA[1618,13] := 890.5168;
   DATA[1618,14] := 1.0;
   DATA[1618,15] := 2.0;
   DATA[1618,16] := 1.0;
   DATA[1618,17] := 1.0;
   DATA[1618,18] := 1.0;
   DATA[1618,19] := 2.0;
   DATA[1618,20] := 148.808;
   DATA[1618,21] := 154.0631;
   DATA[1618,22] := 1.71262;
   DATA[1618,23] := 798.4875;
   DATA[1618,24] := 2.0;
   DATA[1618,25] := 2.0;
   DATA[1618,26] := 7.875737;
   DATA[1618,27] := 142.6045;
   DATA[1618,28] := 262.657;
   DATA[1618,29] := 12.07383;
   DATA[1618,30] := 1.723789;
   DATA[1618,31] := 1.276419;
   DATA[1618,32] := 0.7351407;
   DATA[1618,33] := 0.3082983;
   DATA[1618,34] := 2.0;
   DATA[1618,35] := 250.016;
   DATA[1618,36] := 1.665972;
   DATA[1618,37] := 188.8779;
   DATA[1618,38] := 0.000128152;
   DATA[1618,39] := 1.0;
   DATA[1619,1] := 814.9658;
   DATA[1619,2] := 1.0;
   DATA[1619,3] := 1.0;
   DATA[1619,4] := 262.7211;
   DATA[1619,5] := 8.466612;
   DATA[1619,6] := 319.2771;
   DATA[1619,8] := 1.0;
   DATA[1619,9] := 1.0;
   DATA[1619,10] := 1.0;
   DATA[1619,11] := 19.77079;
   DATA[1619,12] := 2.213881;
   DATA[1619,13] := 890.7172;
   DATA[1619,14] := 1.0;
   DATA[1619,15] := 2.0;
   DATA[1619,16] := 1.0;
   DATA[1619,17] := 1.0;
   DATA[1619,18] := 1.0;
   DATA[1619,19] := 2.0;
   DATA[1619,20] := 148.808;
   DATA[1619,21] := 154.0631;
   DATA[1619,22] := 1.711338;
   DATA[1619,23] := 798.949;
   DATA[1619,24] := 2.0;
   DATA[1619,25] := 2.0;
   DATA[1619,26] := 7.875737;
   DATA[1619,27] := 142.6045;
   DATA[1619,28] := 262.657;
   DATA[1619,29] := 12.07383;
   DATA[1619,30] := 1.724301;
   DATA[1619,31] := 1.286666;
   DATA[1619,32] := 0.7351407;
   DATA[1619,33] := 0.3082983;
   DATA[1619,34] := 2.0;
   DATA[1619,35] := 250.016;
   DATA[1619,36] := 1.665972;
   DATA[1619,37] := 188.8779;
   DATA[1619,38] := 0.000128152;
   DATA[1619,39] := 1.0;
   DATA[1620,1] := 814.9658;
   DATA[1620,2] := 1.0;
   DATA[1620,3] := 1.0;
   DATA[1620,4] := 262.7211;
   DATA[1620,5] := 8.466612;
   DATA[1620,6] := 319.2771;
   DATA[1620,8] := 1.0;
   DATA[1620,9] := 1.0;
   DATA[1620,10] := 1.0;
   DATA[1620,11] := 19.77079;
   DATA[1620,12] := 2.213881;
   DATA[1620,13] := 890.1163;
   DATA[1620,14] := 1.0;
   DATA[1620,15] := 2.0;
   DATA[1620,16] := 1.0;
   DATA[1620,17] := 1.0;
   DATA[1620,18] := 1.0;
   DATA[1620,19] := 2.0;
   DATA[1620,20] := 148.808;
   DATA[1620,21] := 154.0631;
   DATA[1620,22] := 1.711338;
   DATA[1620,23] := 798.9874;
   DATA[1620,24] := 2.0;
   DATA[1620,25] := 2.0;
   DATA[1620,26] := 7.875737;
   DATA[1620,27] := 142.7326;
   DATA[1620,28] := 262.657;
   DATA[1620,29] := 12.07383;
   DATA[1620,30] := 1.724301;
   DATA[1620,31] := 1.291789;
   DATA[1620,32] := 0.7351407;
   DATA[1620,33] := 0.3082983;
   DATA[1620,34] := 2.0;
   DATA[1620,35] := 250.1602;
   DATA[1620,36] := 1.665972;
   DATA[1620,37] := 189.006;
   DATA[1620,38] := 0.000128152;
   DATA[1620,39] := 1.0;
   DATA[1621,1] := 814.9658;
   DATA[1621,2] := 1.0;
   DATA[1621,3] := 1.0;
   DATA[1621,4] := 262.7211;
   DATA[1621,5] := 8.466612;
   DATA[1621,6] := 319.2771;
   DATA[1621,8] := 1.0;
   DATA[1621,9] := 1.0;
   DATA[1621,10] := 1.0;
   DATA[1621,11] := 19.77079;
   DATA[1621,12] := 2.213881;
   DATA[1621,13] := 890.1163;
   DATA[1621,14] := 1.0;
   DATA[1621,15] := 2.0;
   DATA[1621,16] := 1.0;
   DATA[1621,17] := 1.0;
   DATA[1621,18] := 1.0;
   DATA[1621,19] := 2.0;
   DATA[1621,20] := 148.808;
   DATA[1621,21] := 154.0631;
   DATA[1621,22] := 1.711338;
   DATA[1621,23] := 798.9874;
   DATA[1621,24] := 2.0;
   DATA[1621,25] := 2.0;
   DATA[1621,26] := 7.875737;
   DATA[1621,27] := 142.7326;
   DATA[1621,28] := 262.657;
   DATA[1621,29] := 12.07383;
   DATA[1621,30] := 1.724301;
   DATA[1621,31] := 1.291789;
   DATA[1621,32] := 0.7351407;
   DATA[1621,33] := 0.3082983;
   DATA[1621,34] := 2.0;
   DATA[1621,35] := 250.1602;
   DATA[1621,36] := 1.665972;
   DATA[1621,37] := 189.006;
   DATA[1621,38] := 0.000128152;
   DATA[1621,39] := 1.0;
   DATA[1622,1] := 814.8088;
   DATA[1622,2] := 1.0;
   DATA[1622,3] := 1.0;
   DATA[1622,4] := 262.7211;
   DATA[1622,5] := 8.466612;
   DATA[1622,6] := 319.2771;
   DATA[1622,8] := 1.0;
   DATA[1622,9] := 1.0;
   DATA[1622,10] := 1.0;
   DATA[1622,11] := 19.77079;
   DATA[1622,12] := 2.210037;
   DATA[1622,13] := 889.7959;
   DATA[1622,14] := 1.0;
   DATA[1622,15] := 2.0;
   DATA[1622,16] := 1.0;
   DATA[1622,17] := 1.0;
   DATA[1622,18] := 1.0;
   DATA[1622,19] := 2.0;
   DATA[1622,20] := 148.808;
   DATA[1622,21] := 154.0631;
   DATA[1622,22] := 1.711338;
   DATA[1622,23] := 799.3719;
   DATA[1622,24] := 2.0;
   DATA[1622,25] := 2.0;
   DATA[1622,26] := 7.875737;
   DATA[1622,27] := 142.7326;
   DATA[1622,28] := 262.7852;
   DATA[1622,29] := 12.07383;
   DATA[1622,30] := 1.724301;
   DATA[1622,31] := 1.286794;
   DATA[1622,32] := 0.7351407;
   DATA[1622,33] := 0.3082983;
   DATA[1622,34] := 2.0;
   DATA[1622,35] := 250.1602;
   DATA[1622,36] := 1.665972;
   DATA[1622,37] := 189.006;
   DATA[1622,38] := 0.000128152;
   DATA[1622,39] := 1.0;
   DATA[1623,1] := 814.6125;
   DATA[1623,2] := 1.0;
   DATA[1623,3] := 1.0;
   DATA[1623,4] := 262.7211;
   DATA[1623,5] := 8.466612;
   DATA[1623,6] := 319.2771;
   DATA[1623,8] := 1.0;
   DATA[1623,9] := 1.0;
   DATA[1623,10] := 1.0;
   DATA[1623,11] := 19.77079;
   DATA[1623,12] := 2.209397;
   DATA[1623,13] := 889.1951;
   DATA[1623,14] := 1.0;
   DATA[1623,15] := 2.0;
   DATA[1623,16] := 1.0;
   DATA[1623,17] := 1.0;
   DATA[1623,18] := 1.0;
   DATA[1623,19] := 2.0;
   DATA[1623,20] := 148.808;
   DATA[1623,21] := 154.0631;
   DATA[1623,22] := 1.711338;
   DATA[1623,23] := 799.1797;
   DATA[1623,24] := 2.0;
   DATA[1623,25] := 2.0;
   DATA[1623,26] := 7.875737;
   DATA[1623,27] := 142.7326;
   DATA[1623,28] := 262.7852;
   DATA[1623,29] := 12.07383;
   DATA[1623,30] := 1.724301;
   DATA[1623,31] := 1.290637;
   DATA[1623,32] := 0.7351407;
   DATA[1623,33] := 0.3082983;
   DATA[1623,34] := 2.0;
   DATA[1623,35] := 250.1602;
   DATA[1623,36] := 1.665972;
   DATA[1623,37] := 189.1823;
   DATA[1623,38] := 0.000128152;
   DATA[1623,39] := 1.0;
   DATA[1624,1] := 814.534;
   DATA[1624,2] := 1.0;
   DATA[1624,3] := 1.0;
   DATA[1624,4] := 262.7211;
   DATA[1624,5] := 8.466612;
   DATA[1624,6] := 319.2771;
   DATA[1624,8] := 1.0;
   DATA[1624,9] := 1.0;
   DATA[1624,10] := 1.0;
   DATA[1624,11] := 19.80601;
   DATA[1624,12] := 2.209397;
   DATA[1624,13] := 888.8346;
   DATA[1624,14] := 1.0;
   DATA[1624,15] := 2.0;
   DATA[1624,16] := 1.0;
   DATA[1624,17] := 1.0;
   DATA[1624,18] := 1.0;
   DATA[1624,19] := 2.0;
   DATA[1624,20] := 148.808;
   DATA[1624,21] := 153.858;
   DATA[1624,22] := 1.711338;
   DATA[1624,23] := 798.8336;
   DATA[1624,24] := 2.0;
   DATA[1624,25] := 2.0;
   DATA[1624,26] := 7.875737;
   DATA[1624,27] := 142.7326;
   DATA[1624,28] := 262.7852;
   DATA[1624,29] := 12.07383;
   DATA[1624,30] := 1.724301;
   DATA[1624,31] := 1.292046;
   DATA[1624,32] := 0.7351407;
   DATA[1624,33] := 0.3082983;
   DATA[1624,34] := 2.0;
   DATA[1624,35] := 250.1602;
   DATA[1624,36] := 1.665972;
   DATA[1624,37] := 189.1823;
   DATA[1624,38] := 0.000128152;
   DATA[1624,39] := 1.0;
   DATA[1625,1] := 814.1807;
   DATA[1625,2] := 1.0;
   DATA[1625,3] := 1.0;
   DATA[1625,4] := 262.7211;
   DATA[1625,5] := 8.466612;
   DATA[1625,6] := 319.2771;
   DATA[1625,8] := 1.0;
   DATA[1625,9] := 1.0;
   DATA[1625,10] := 1.0;
   DATA[1625,11] := 19.80601;
   DATA[1625,12] := 2.209397;
   DATA[1625,13] := 888.4341;
   DATA[1625,14] := 1.0;
   DATA[1625,15] := 2.0;
   DATA[1625,16] := 1.0;
   DATA[1625,17] := 1.0;
   DATA[1625,18] := 1.0;
   DATA[1625,19] := 2.0;
   DATA[1625,20] := 148.808;
   DATA[1625,21] := 153.858;
   DATA[1625,22] := 1.711338;
   DATA[1625,23] := 798.7952;
   DATA[1625,24] := 2.0;
   DATA[1625,25] := 2.0;
   DATA[1625,26] := 7.875737;
   DATA[1625,27] := 142.7326;
   DATA[1625,28] := 262.7852;
   DATA[1625,29] := 12.15073;
   DATA[1625,30] := 1.724301;
   DATA[1625,31] := 1.28167;
   DATA[1625,32] := 0.7351407;
   DATA[1625,33] := 0.3082983;
   DATA[1625,34] := 2.0;
   DATA[1625,35] := 250.1602;
   DATA[1625,36] := 1.665972;
   DATA[1625,37] := 189.1823;
   DATA[1625,38] := 0.000128152;
   DATA[1625,39] := 1.0;
   DATA[1626,1] := 814.1415;
   DATA[1626,2] := 1.0;
   DATA[1626,3] := 1.0;
   DATA[1626,4] := 262.5288;
   DATA[1626,5] := 8.466612;
   DATA[1626,6] := 319.2771;
   DATA[1626,8] := 1.0;
   DATA[1626,9] := 1.0;
   DATA[1626,10] := 1.0;
   DATA[1626,11] := 19.80601;
   DATA[1626,12] := 2.209397;
   DATA[1626,13] := 887.9935;
   DATA[1626,14] := 1.0;
   DATA[1626,15] := 2.0;
   DATA[1626,16] := 1.0;
   DATA[1626,17] := 1.0;
   DATA[1626,18] := 1.0;
   DATA[1626,19] := 2.0;
   DATA[1626,20] := 148.808;
   DATA[1626,21] := 153.858;
   DATA[1626,22] := 1.711338;
   DATA[1626,23] := 798.5645;
   DATA[1626,24] := 2.0;
   DATA[1626,25] := 2.0;
   DATA[1626,26] := 7.876058;
   DATA[1626,27] := 142.7326;
   DATA[1626,28] := 262.7852;
   DATA[1626,29] := 12.15073;
   DATA[1626,30] := 1.724301;
   DATA[1626,31] := 1.273216;
   DATA[1626,32] := 0.7351407;
   DATA[1626,33] := 0.3082983;
   DATA[1626,34] := 2.0;
   DATA[1626,35] := 250.1602;
   DATA[1626,36] := 1.665972;
   DATA[1626,37] := 189.1823;
   DATA[1626,38] := 0.000128152;
   DATA[1626,39] := 1.0;
   DATA[1627,1] := 814.5732;
   DATA[1627,2] := 1.0;
   DATA[1627,3] := 1.0;
   DATA[1627,4] := 262.5288;
   DATA[1627,5] := 8.466612;
   DATA[1627,6] := 319.2771;
   DATA[1627,8] := 1.0;
   DATA[1627,9] := 1.0;
   DATA[1627,10] := 1.0;
   DATA[1627,11] := 19.8028;
   DATA[1627,12] := 2.209397;
   DATA[1627,13] := 887.7131;
   DATA[1627,14] := 1.0;
   DATA[1627,15] := 2.0;
   DATA[1627,16] := 1.0;
   DATA[1627,17] := 1.0;
   DATA[1627,18] := 1.0;
   DATA[1627,19] := 2.0;
   DATA[1627,20] := 148.808;
   DATA[1627,21] := 154.0374;
   DATA[1627,22] := 1.712748;
   DATA[1627,23] := 798.5645;
   DATA[1627,24] := 2.0;
   DATA[1627,25] := 2.0;
   DATA[1627,26] := 7.877019;
   DATA[1627,27] := 142.7326;
   DATA[1627,28] := 262.7852;
   DATA[1627,29] := 12.15073;
   DATA[1627,30] := 1.724301;
   DATA[1627,31] := 1.271679;
   DATA[1627,32] := 0.7351407;
   DATA[1627,33] := 0.3082983;
   DATA[1627,34] := 2.0;
   DATA[1627,35] := 250.1602;
   DATA[1627,36] := 1.665972;
   DATA[1627,37] := 189.0861;
   DATA[1627,38] := 0.000128152;
   DATA[1627,39] := 1.0;
   DATA[1628,1] := 814.3377;
   DATA[1628,2] := 1.0;
   DATA[1628,3] := 1.0;
   DATA[1628,4] := 262.5288;
   DATA[1628,5] := 8.466612;
   DATA[1628,6] := 319.2771;
   DATA[1628,8] := 1.0;
   DATA[1628,9] := 1.0;
   DATA[1628,10] := 1.0;
   DATA[1628,11] := 19.74838;
   DATA[1628,12] := 2.209397;
   DATA[1628,13] := 887.5128;
   DATA[1628,14] := 1.0;
   DATA[1628,15] := 2.0;
   DATA[1628,16] := 1.0;
   DATA[1628,17] := 1.0;
   DATA[1628,18] := 1.0;
   DATA[1628,19] := 2.0;
   DATA[1628,20] := 148.808;
   DATA[1628,21] := 154.0374;
   DATA[1628,22] := 1.712748;
   DATA[1628,23] := 798.7952;
   DATA[1628,24] := 2.0;
   DATA[1628,25] := 2.0;
   DATA[1628,26] := 7.877019;
   DATA[1628,27] := 142.7326;
   DATA[1628,28] := 262.7852;
   DATA[1628,29] := 12.15073;
   DATA[1628,30] := 1.72507;
   DATA[1628,31] := 1.271679;
   DATA[1628,32] := 0.7351407;
   DATA[1628,33] := 0.3082983;
   DATA[1628,34] := 2.0;
   DATA[1628,35] := 250.1602;
   DATA[1628,36] := 1.665972;
   DATA[1628,37] := 189.0381;
   DATA[1628,38] := 0.000128152;
   DATA[1628,39] := 1.0;
   DATA[1629,1] := 813.8275;
   DATA[1629,2] := 1.0;
   DATA[1629,3] := 1.0;
   DATA[1629,4] := 262.5288;
   DATA[1629,5] := 8.466612;
   DATA[1629,6] := 319.2771;
   DATA[1629,8] := 1.0;
   DATA[1629,9] := 1.0;
   DATA[1629,10] := 1.0;
   DATA[1629,11] := 19.74838;
   DATA[1629,12] := 2.209397;
   DATA[1629,13] := 886.7518;
   DATA[1629,14] := 1.0;
   DATA[1629,15] := 2.0;
   DATA[1629,16] := 1.0;
   DATA[1629,17] := 1.0;
   DATA[1629,18] := 1.0;
   DATA[1629,19] := 2.0;
   DATA[1629,20] := 148.808;
   DATA[1629,21] := 154.1656;
   DATA[1629,22] := 1.712748;
   DATA[1629,23] := 799.4489;
   DATA[1629,24] := 2.0;
   DATA[1629,25] := 2.0;
   DATA[1629,26] := 7.877019;
   DATA[1629,27] := 142.7326;
   DATA[1629,28] := 262.7852;
   DATA[1629,29] := 12.15073;
   DATA[1629,30] := 1.72507;
   DATA[1629,31] := 1.263866;
   DATA[1629,32] := 0.7351407;
   DATA[1629,33] := 0.3082983;
   DATA[1629,34] := 2.0;
   DATA[1629,35] := 250.1602;
   DATA[1629,36] := 1.665972;
   DATA[1629,37] := 189.0381;
   DATA[1629,38] := 0.000128152;
   DATA[1629,39] := 1.0;
   DATA[1630,1] := 814.1022;
   DATA[1630,2] := 1.0;
   DATA[1630,3] := 1.0;
   DATA[1630,4] := 262.5288;
   DATA[1630,5] := 8.466612;
   DATA[1630,6] := 319.2771;
   DATA[1630,8] := 1.0;
   DATA[1630,9] := 1.0;
   DATA[1630,10] := 1.0;
   DATA[1630,11] := 19.77079;
   DATA[1630,12] := 2.2126;
   DATA[1630,13] := 886.5516;
   DATA[1630,14] := 1.0;
   DATA[1630,15] := 2.0;
   DATA[1630,16] := 1.0;
   DATA[1630,17] := 1.0;
   DATA[1630,18] := 1.0;
   DATA[1630,19] := 2.0;
   DATA[1630,20] := 148.808;
   DATA[1630,21] := 154.1656;
   DATA[1630,22] := 1.712748;
   DATA[1630,23] := 799.4104;
   DATA[1630,24] := 2.0;
   DATA[1630,25] := 2.0;
   DATA[1630,26] := 7.877019;
   DATA[1630,27] := 142.7326;
   DATA[1630,28] := 262.7852;
   DATA[1630,29] := 12.15073;
   DATA[1630,30] := 1.72507;
   DATA[1630,31] := 1.262329;
   DATA[1630,32] := 0.7351407;
   DATA[1630,33] := 0.3082983;
   DATA[1630,34] := 2.0;
   DATA[1630,35] := 250.1602;
   DATA[1630,36] := 1.665972;
   DATA[1630,37] := 189.0381;
   DATA[1630,38] := 0.000128152;
   DATA[1630,39] := 1.0;
   DATA[1631,1] := 814.3377;
   DATA[1631,2] := 1.0;
   DATA[1631,3] := 1.0;
   DATA[1631,4] := 262.5288;
   DATA[1631,5] := 8.466612;
   DATA[1631,6] := 319.2771;
   DATA[1631,8] := 1.0;
   DATA[1631,9] := 1.0;
   DATA[1631,10] := 1.0;
   DATA[1631,11] := 19.77079;
   DATA[1631,12] := 2.2126;
   DATA[1631,13] := 886.6317;
   DATA[1631,14] := 1.0;
   DATA[1631,15] := 2.0;
   DATA[1631,16] := 1.0;
   DATA[1631,17] := 1.0;
   DATA[1631,18] := 1.0;
   DATA[1631,19] := 2.0;
   DATA[1631,20] := 148.808;
   DATA[1631,21] := 154.1656;
   DATA[1631,22] := 1.712748;
   DATA[1631,23] := 799.2181;
   DATA[1631,24] := 2.0;
   DATA[1631,25] := 2.0;
   DATA[1631,26] := 7.877019;
   DATA[1631,27] := 142.7326;
   DATA[1631,28] := 262.7852;
   DATA[1631,29] := 12.15073;
   DATA[1631,30] := 1.72507;
   DATA[1631,31] := 1.270783;
   DATA[1631,32] := 0.7351407;
   DATA[1631,33] := 0.3082983;
   DATA[1631,34] := 2.0;
   DATA[1631,35] := 250.1602;
   DATA[1631,36] := 1.665972;
   DATA[1631,37] := 189.0381;
   DATA[1631,38] := 0.000128152;
   DATA[1631,39] := 1.0;
   DATA[1632,1] := 814.377;
   DATA[1632,2] := 1.0;
   DATA[1632,3] := 1.0;
   DATA[1632,4] := 262.5288;
   DATA[1632,5] := 8.46501;
   DATA[1632,6] := 319.2771;
   DATA[1632,8] := 1.0;
   DATA[1632,9] := 1.0;
   DATA[1632,10] := 1.0;
   DATA[1632,11] := 19.77079;
   DATA[1632,12] := 2.2126;
   DATA[1632,13] := 886.0308;
   DATA[1632,14] := 1.0;
   DATA[1632,15] := 2.0;
   DATA[1632,16] := 1.0;
   DATA[1632,17] := 1.0;
   DATA[1632,18] := 1.0;
   DATA[1632,19] := 2.0;
   DATA[1632,20] := 148.808;
   DATA[1632,21] := 154.1656;
   DATA[1632,22] := 1.712235;
   DATA[1632,23] := 799.4489;
   DATA[1632,24] := 2.0;
   DATA[1632,25] := 2.0;
   DATA[1632,26] := 7.876058;
   DATA[1632,27] := 142.7326;
   DATA[1632,28] := 262.7852;
   DATA[1632,29] := 12.15073;
   DATA[1632,30] := 1.72507;
   DATA[1632,31] := 1.271935;
   DATA[1632,32] := 0.7351407;
   DATA[1632,33] := 0.3082983;
   DATA[1632,34] := 2.0;
   DATA[1632,35] := 250.1602;
   DATA[1632,36] := 1.665972;
   DATA[1632,37] := 189.0381;
   DATA[1632,38] := 0.000128152;
   DATA[1632,39] := 1.0;
   DATA[1633,1] := 814.4162;
   DATA[1633,2] := 1.0;
   DATA[1633,3] := 1.0;
   DATA[1633,4] := 262.5288;
   DATA[1633,5] := 8.46501;
   DATA[1633,6] := 319.2771;
   DATA[1633,8] := 1.0;
   DATA[1633,9] := 1.0;
   DATA[1633,10] := 1.0;
   DATA[1633,11] := 19.77079;
   DATA[1633,12] := 2.2126;
   DATA[1633,13] := 885.7505;
   DATA[1633,14] := 1.0;
   DATA[1633,15] := 2.0;
   DATA[1633,16] := 1.0;
   DATA[1633,17] := 1.0;
   DATA[1633,18] := 1.0;
   DATA[1633,19] := 2.0;
   DATA[1633,20] := 148.808;
   DATA[1633,21] := 154.1656;
   DATA[1633,22] := 1.711466;
   DATA[1633,23] := 799.4104;
   DATA[1633,24] := 2.0;
   DATA[1633,25] := 2.0;
   DATA[1633,26] := 7.876058;
   DATA[1633,27] := 142.7326;
   DATA[1633,28] := 262.7852;
   DATA[1633,29] := 12.15073;
   DATA[1633,30] := 1.72507;
   DATA[1633,31] := 1.280389;
   DATA[1633,32] := 0.7351407;
   DATA[1633,33] := 0.3082983;
   DATA[1633,34] := 2.0;
   DATA[1633,35] := 250.1602;
   DATA[1633,36] := 1.665972;
   DATA[1633,37] := 189.0381;
   DATA[1633,38] := 0.000128152;
   DATA[1633,39] := 1.0;
   DATA[1634,1] := 814.2985;
   DATA[1634,2] := 1.0;
   DATA[1634,3] := 1.0;
   DATA[1634,4] := 262.5288;
   DATA[1634,5] := 8.46501;
   DATA[1634,6] := 319.2771;
   DATA[1634,8] := 1.0;
   DATA[1634,9] := 1.0;
   DATA[1634,10] := 1.0;
   DATA[1634,11] := 19.77079;
   DATA[1634,12] := 2.213624;
   DATA[1634,13] := 885.1497;
   DATA[1634,14] := 1.0;
   DATA[1634,15] := 2.0;
   DATA[1634,16] := 1.0;
   DATA[1634,17] := 1.0;
   DATA[1634,18] := 1.0;
   DATA[1634,19] := 2.0;
   DATA[1634,20] := 148.808;
   DATA[1634,21] := 154.1656;
   DATA[1634,22] := 1.711466;
   DATA[1634,23] := 799.4489;
   DATA[1634,24] := 2.0;
   DATA[1634,25] := 2.0;
   DATA[1634,26] := 7.876058;
   DATA[1634,27] := 142.7326;
   DATA[1634,28] := 262.7852;
   DATA[1634,29] := 12.15073;
   DATA[1634,30] := 1.72507;
   DATA[1634,31] := 1.281286;
   DATA[1634,32] := 0.7351407;
   DATA[1634,33] := 0.3082983;
   DATA[1634,34] := 2.0;
   DATA[1634,35] := 250.1602;
   DATA[1634,36] := 1.665972;
   DATA[1634,37] := 189.0381;
   DATA[1634,38] := 0.000128152;
   DATA[1634,39] := 1.0;
   DATA[1635,1] := 814.0237;
   DATA[1635,2] := 1.0;
   DATA[1635,3] := 1.0;
   DATA[1635,4] := 262.5288;
   DATA[1635,5] := 8.46501;
   DATA[1635,6] := 319.2771;
   DATA[1635,8] := 1.0;
   DATA[1635,9] := 1.0;
   DATA[1635,10] := 1.0;
   DATA[1635,11] := 19.77079;
   DATA[1635,12] := 2.213624;
   DATA[1635,13] := 884.1483;
   DATA[1635,14] := 1.0;
   DATA[1635,15] := 2.0;
   DATA[1635,16] := 1.0;
   DATA[1635,17] := 1.0;
   DATA[1635,18] := 1.0;
   DATA[1635,19] := 2.0;
   DATA[1635,20] := 148.808;
   DATA[1635,21] := 154.1656;
   DATA[1635,22] := 1.711466;
   DATA[1635,23] := 799.5258;
   DATA[1635,24] := 2.0;
   DATA[1635,25] := 2.0;
   DATA[1635,26] := 7.876058;
   DATA[1635,27] := 142.7326;
   DATA[1635,28] := 262.7852;
   DATA[1635,29] := 12.15073;
   DATA[1635,30] := 1.72507;
   DATA[1635,31] := 1.271551;
   DATA[1635,32] := 0.7351407;
   DATA[1635,33] := 0.3082983;
   DATA[1635,34] := 2.0;
   DATA[1635,35] := 250.1602;
   DATA[1635,36] := 1.665972;
   DATA[1635,37] := 189.0381;
   DATA[1635,38] := 0.000128152;
   DATA[1635,39] := 1.0;
   DATA[1636,1] := 813.9452;
   DATA[1636,2] := 1.0;
   DATA[1636,3] := 1.0;
   DATA[1636,4] := 262.5288;
   DATA[1636,5] := 8.46501;
   DATA[1636,6] := 319.2771;
   DATA[1636,8] := 1.0;
   DATA[1636,9] := 1.0;
   DATA[1636,10] := 1.0;
   DATA[1636,11] := 19.77079;
   DATA[1636,12] := 2.213624;
   DATA[1636,13] := 883.9481;
   DATA[1636,14] := 1.0;
   DATA[1636,15] := 2.0;
   DATA[1636,16] := 1.0;
   DATA[1636,17] := 1.0;
   DATA[1636,18] := 1.0;
   DATA[1636,19] := 2.0;
   DATA[1636,20] := 148.808;
   DATA[1636,21] := 154.1656;
   DATA[1636,22] := 1.711466;
   DATA[1636,23] := 799.4104;
   DATA[1636,24] := 2.0;
   DATA[1636,25] := 2.0;
   DATA[1636,26] := 7.876058;
   DATA[1636,27] := 142.7326;
   DATA[1636,28] := 262.7852;
   DATA[1636,29] := 12.15073;
   DATA[1636,30] := 1.72507;
   DATA[1636,31] := 1.271551;
   DATA[1636,32] := 0.7351407;
   DATA[1636,33] := 0.3082983;
   DATA[1636,34] := 2.0;
   DATA[1636,35] := 250.1602;
   DATA[1636,36] := 1.665972;
   DATA[1636,37] := 188.974;
   DATA[1636,38] := 0.000128152;
   DATA[1636,39] := 1.0;
   DATA[1637,1] := 813.9059;
   DATA[1637,2] := 1.0;
   DATA[1637,3] := 1.0;
   DATA[1637,4] := 262.5288;
   DATA[1637,5] := 8.46501;
   DATA[1637,6] := 319.2771;
   DATA[1637,8] := 1.0;
   DATA[1637,9] := 1.0;
   DATA[1637,10] := 1.0;
   DATA[1637,11] := 19.77079;
   DATA[1637,12] := 2.213624;
   DATA[1637,13] := 883.5074;
   DATA[1637,14] := 1.0;
   DATA[1637,15] := 2.0;
   DATA[1637,16] := 1.0;
   DATA[1637,17] := 1.0;
   DATA[1637,18] := 1.0;
   DATA[1637,19] := 2.0;
   DATA[1637,20] := 148.808;
   DATA[1637,21] := 154.1656;
   DATA[1637,22] := 1.712363;
   DATA[1637,23] := 799.2181;
   DATA[1637,24] := 2.0;
   DATA[1637,25] := 2.0;
   DATA[1637,26] := 7.876058;
   DATA[1637,27] := 142.7326;
   DATA[1637,28] := 262.7852;
   DATA[1637,29] := 12.15073;
   DATA[1637,30] := 1.72507;
   DATA[1637,31] := 1.273345;
   DATA[1637,32] := 0.7351407;
   DATA[1637,33] := 0.3082983;
   DATA[1637,34] := 2.0;
   DATA[1637,35] := 250.1602;
   DATA[1637,36] := 1.665972;
   DATA[1637,37] := 188.974;
   DATA[1637,38] := 0.000128152;
   DATA[1637,39] := 1.0;
   DATA[1638,1] := 813.9844;
   DATA[1638,2] := 1.0;
   DATA[1638,3] := 1.0;
   DATA[1638,4] := 262.5288;
   DATA[1638,5] := 8.46501;
   DATA[1638,6] := 319.2771;
   DATA[1638,8] := 1.0;
   DATA[1638,9] := 1.0;
   DATA[1638,10] := 1.0;
   DATA[1638,11] := 19.77079;
   DATA[1638,12] := 2.213624;
   DATA[1638,13] := 883.2271;
   DATA[1638,14] := 1.0;
   DATA[1638,15] := 2.0;
   DATA[1638,16] := 1.0;
   DATA[1638,17] := 1.0;
   DATA[1638,18] := 1.0;
   DATA[1638,19] := 2.0;
   DATA[1638,20] := 148.808;
   DATA[1638,21] := 154.1656;
   DATA[1638,22] := 1.713261;
   DATA[1638,23] := 799.5642;
   DATA[1638,24] := 2.0;
   DATA[1638,25] := 2.0;
   DATA[1638,26] := 7.876058;
   DATA[1638,27] := 142.7326;
   DATA[1638,28] := 262.7852;
   DATA[1638,29] := 11.92002;
   DATA[1638,30] := 1.72507;
   DATA[1638,31] := 1.288843;
   DATA[1638,32] := 0.7351407;
   DATA[1638,33] := 0.3082983;
   DATA[1638,34] := 2.0;
   DATA[1638,35] := 250.1602;
   DATA[1638,36] := 1.665972;
   DATA[1638,37] := 188.974;
   DATA[1638,38] := 0.000128152;
   DATA[1638,39] := 1.0;
   DATA[1639,1] := 813.8275;
   DATA[1639,2] := 1.0;
   DATA[1639,3] := 1.0;
   DATA[1639,4] := 262.5288;
   DATA[1639,5] := 8.46501;
   DATA[1639,6] := 319.2771;
   DATA[1639,8] := 1.0;
   DATA[1639,9] := 1.0;
   DATA[1639,10] := 1.0;
   DATA[1639,11] := 19.7996;
   DATA[1639,12] := 2.213624;
   DATA[1639,13] := 882.426;
   DATA[1639,14] := 1.0;
   DATA[1639,15] := 2.0;
   DATA[1639,16] := 1.0;
   DATA[1639,17] := 1.0;
   DATA[1639,18] := 1.0;
   DATA[1639,19] := 2.0;
   DATA[1639,20] := 148.808;
   DATA[1639,21] := 154.1656;
   DATA[1639,22] := 1.713901;
   DATA[1639,23] := 799.718;
   DATA[1639,24] := 2.0;
   DATA[1639,25] := 2.0;
   DATA[1639,26] := 7.876058;
   DATA[1639,27] := 142.7326;
   DATA[1639,28] := 262.7852;
   DATA[1639,29] := 11.92002;
   DATA[1639,30] := 1.72507;
   DATA[1639,31] := 1.291918;
   DATA[1639,32] := 0.7351407;
   DATA[1639,33] := 0.3082983;
   DATA[1639,34] := 2.0;
   DATA[1639,35] := 250.3044;
   DATA[1639,36] := 1.665972;
   DATA[1639,37] := 188.974;
   DATA[1639,38] := 0.000128152;
   DATA[1639,39] := 1.0;
   DATA[1640,1] := 814.22;
   DATA[1640,2] := 1.0;
   DATA[1640,3] := 1.0;
   DATA[1640,4] := 262.5288;
   DATA[1640,5] := 8.46501;
   DATA[1640,6] := 319.2771;
   DATA[1640,8] := 1.0;
   DATA[1640,9] := 1.0;
   DATA[1640,10] := 1.0;
   DATA[1640,11] := 19.7996;
   DATA[1640,12] := 2.213624;
   DATA[1640,13] := 881.9454;
   DATA[1640,14] := 1.0;
   DATA[1640,15] := 2.0;
   DATA[1640,16] := 1.0;
   DATA[1640,17] := 1.0;
   DATA[1640,18] := 1.0;
   DATA[1640,19] := 2.0;
   DATA[1640,20] := 148.808;
   DATA[1640,21] := 154.1656;
   DATA[1640,22] := 1.715183;
   DATA[1640,23] := 799.7565;
   DATA[1640,24] := 2.0;
   DATA[1640,25] := 2.0;
   DATA[1640,26] := 7.876058;
   DATA[1640,27] := 142.8095;
   DATA[1640,28] := 262.7852;
   DATA[1640,29] := 11.92002;
   DATA[1640,30] := 1.72507;
   DATA[1640,31] := 1.29243;
   DATA[1640,32] := 0.7351407;
   DATA[1640,33] := 0.3082983;
   DATA[1640,34] := 2.0;
   DATA[1640,35] := 250.3044;
   DATA[1640,36] := 1.665972;
   DATA[1640,37] := 188.974;
   DATA[1640,38] := 0.000128152;
   DATA[1640,39] := 1.0;
   DATA[1641,1] := 814.22;
   DATA[1641,2] := 1.0;
   DATA[1641,3] := 1.0;
   DATA[1641,4] := 262.5288;
   DATA[1641,5] := 8.46501;
   DATA[1641,6] := 319.2771;
   DATA[1641,8] := 1.0;
   DATA[1641,9] := 1.0;
   DATA[1641,10] := 1.0;
   DATA[1641,11] := 19.76439;
   DATA[1641,12] := 2.213624;
   DATA[1641,13] := 881.3445;
   DATA[1641,14] := 1.0;
   DATA[1641,15] := 2.0;
   DATA[1641,16] := 1.0;
   DATA[1641,17] := 1.0;
   DATA[1641,18] := 1.0;
   DATA[1641,19] := 2.0;
   DATA[1641,20] := 148.808;
   DATA[1641,21] := 154.1656;
   DATA[1641,22] := 1.715183;
   DATA[1641,23] := 799.6411;
   DATA[1641,24] := 2.0;
   DATA[1641,25] := 2.0;
   DATA[1641,26] := 7.876058;
   DATA[1641,27] := 142.9121;
   DATA[1641,28] := 262.7852;
   DATA[1641,29] := 12.03538;
   DATA[1641,30] := 1.723532;
   DATA[1641,31] := 1.29243;
   DATA[1641,32] := 0.7351407;
   DATA[1641,33] := 0.3082983;
   DATA[1641,34] := 2.0;
   DATA[1641,35] := 250.3044;
   DATA[1641,36] := 1.665972;
   DATA[1641,37] := 188.974;
   DATA[1641,38] := 0.000128152;
   DATA[1641,39] := 1.0;
   DATA[1642,1] := 814.3377;
   DATA[1642,2] := 1.0;
   DATA[1642,3] := 1.0;
   DATA[1642,4] := 262.5288;
   DATA[1642,5] := 8.46501;
   DATA[1642,6] := 319.2771;
   DATA[1642,8] := 1.0;
   DATA[1642,9] := 1.0;
   DATA[1642,10] := 1.0;
   DATA[1642,11] := 19.69396;
   DATA[1642,12] := 2.213624;
   DATA[1642,13] := 880.7838;
   DATA[1642,14] := 1.0;
   DATA[1642,15] := 2.0;
   DATA[1642,16] := 1.0;
   DATA[1642,17] := 1.0;
   DATA[1642,18] := 1.0;
   DATA[1642,19] := 2.0;
   DATA[1642,20] := 148.808;
   DATA[1642,21] := 154.1656;
   DATA[1642,22] := 1.715183;
   DATA[1642,23] := 799.4489;
   DATA[1642,24] := 2.0;
   DATA[1642,25] := 2.0;
   DATA[1642,26] := 7.876058;
   DATA[1642,27] := 142.9121;
   DATA[1642,28] := 262.7852;
   DATA[1642,29] := 12.03538;
   DATA[1642,30] := 1.723532;
   DATA[1642,31] := 1.283207;
   DATA[1642,32] := 0.7351407;
   DATA[1642,33] := 0.3082983;
   DATA[1642,34] := 2.0;
   DATA[1642,35] := 250.3044;
   DATA[1642,36] := 1.665972;
   DATA[1642,37] := 189.0541;
   DATA[1642,38] := 0.000128152;
   DATA[1642,39] := 1.0;
   DATA[1643,1] := 814.7695;
   DATA[1643,2] := 1.0;
   DATA[1643,3] := 1.0;
   DATA[1643,4] := 262.5288;
   DATA[1643,5] := 8.466932;
   DATA[1643,6] := 319.2771;
   DATA[1643,8] := 1.0;
   DATA[1643,9] := 1.0;
   DATA[1643,10] := 1.0;
   DATA[1643,11] := 19.69076;
   DATA[1643,12] := 2.213624;
   DATA[1643,13] := 880.5835;
   DATA[1643,14] := 1.0;
   DATA[1643,15] := 2.0;
   DATA[1643,16] := 1.0;
   DATA[1643,17] := 1.0;
   DATA[1643,18] := 1.0;
   DATA[1643,19] := 2.0;
   DATA[1643,20] := 148.808;
   DATA[1643,21] := 154.1656;
   DATA[1643,22] := 1.715183;
   DATA[1643,23] := 799.3719;
   DATA[1643,24] := 2.0;
   DATA[1643,25] := 2.0;
   DATA[1643,26] := 7.876058;
   DATA[1643,27] := 142.9121;
   DATA[1643,28] := 262.7852;
   DATA[1643,29] := 12.03538;
   DATA[1643,30] := 1.723532;
   DATA[1643,31] := 1.271935;
   DATA[1643,32] := 0.7351407;
   DATA[1643,33] := 0.3082983;
   DATA[1643,34] := 2.0;
   DATA[1643,35] := 250.2243;
   DATA[1643,36] := 1.665972;
   DATA[1643,37] := 189.0541;
   DATA[1643,38] := 0.000128152;
   DATA[1643,39] := 1.0;
   DATA[1644,1] := 814.6125;
   DATA[1644,2] := 1.0;
   DATA[1644,3] := 1.0;
   DATA[1644,4] := 262.5288;
   DATA[1644,5] := 8.466932;
   DATA[1644,6] := 319.2771;
   DATA[1644,8] := 1.0;
   DATA[1644,9] := 1.0;
   DATA[1644,10] := 1.0;
   DATA[1644,11] := 19.69076;
   DATA[1644,12] := 2.213624;
   DATA[1644,13] := 879.9427;
   DATA[1644,14] := 1.0;
   DATA[1644,15] := 2.0;
   DATA[1644,16] := 1.0;
   DATA[1644,17] := 1.0;
   DATA[1644,18] := 1.0;
   DATA[1644,19] := 2.0;
   DATA[1644,20] := 148.808;
   DATA[1644,21] := 154.1656;
   DATA[1644,22] := 1.715183;
   DATA[1644,23] := 799.6411;
   DATA[1644,24] := 2.0;
   DATA[1644,25] := 2.0;
   DATA[1644,26] := 7.876058;
   DATA[1644,27] := 142.9121;
   DATA[1644,28] := 262.7852;
   DATA[1644,29] := 12.03538;
   DATA[1644,30] := 1.723532;
   DATA[1644,31] := 1.276162;
   DATA[1644,32] := 0.7351407;
   DATA[1644,33] := 0.3082983;
   DATA[1644,34] := 2.0;
   DATA[1644,35] := 250.1442;
   DATA[1644,36] := 1.521802;
   DATA[1644,37] := 189.0541;
   DATA[1644,38] := 0.000128152;
   DATA[1644,39] := 1.0;
   DATA[1645,1] := 814.2985;
   DATA[1645,2] := 1.0;
   DATA[1645,3] := 1.0;
   DATA[1645,4] := 262.7211;
   DATA[1645,5] := 8.466932;
   DATA[1645,6] := 319.2771;
   DATA[1645,8] := 1.0;
   DATA[1645,9] := 1.0;
   DATA[1645,10] := 1.0;
   DATA[1645,11] := 19.74198;
   DATA[1645,12] := 2.213624;
   DATA[1645,13] := 879.7424;
   DATA[1645,14] := 1.0;
   DATA[1645,15] := 2.0;
   DATA[1645,16] := 1.0;
   DATA[1645,17] := 1.0;
   DATA[1645,18] := 1.0;
   DATA[1645,19] := 2.0;
   DATA[1645,20] := 148.808;
   DATA[1645,21] := 154.1656;
   DATA[1645,22] := 1.715183;
   DATA[1645,23] := 799.3719;
   DATA[1645,24] := 2.0;
   DATA[1645,25] := 2.0;
   DATA[1645,26] := 7.876058;
   DATA[1645,27] := 142.9121;
   DATA[1645,28] := 262.7852;
   DATA[1645,29] := 12.03538;
   DATA[1645,30] := 1.723532;
   DATA[1645,31] := 1.277187;
   DATA[1645,32] := 0.7355248;
   DATA[1645,33] := 0.3082983;
   DATA[1645,34] := 2.0;
   DATA[1645,35] := 250.0801;
   DATA[1645,36] := 1.521802;
   DATA[1645,37] := 189.0541;
   DATA[1645,38] := 0.000128152;
   DATA[1645,39] := 1.0;
   DATA[1646,1] := 814.1807;
   DATA[1646,2] := 1.0;
   DATA[1646,3] := 1.0;
   DATA[1646,4] := 262.7211;
   DATA[1646,5] := 8.466932;
   DATA[1646,6] := 319.2771;
   DATA[1646,8] := 1.0;
   DATA[1646,9] := 1.0;
   DATA[1646,10] := 1.0;
   DATA[1646,11] := 19.74198;
   DATA[1646,12] := 2.213624;
   DATA[1646,13] := 879.3018;
   DATA[1646,14] := 1.0;
   DATA[1646,15] := 2.0;
   DATA[1646,16] := 1.0;
   DATA[1646,17] := 1.0;
   DATA[1646,18] := 1.0;
   DATA[1646,19] := 2.0;
   DATA[1646,20] := 148.808;
   DATA[1646,21] := 154.1656;
   DATA[1646,22] := 1.716208;
   DATA[1646,23] := 799.4104;
   DATA[1646,24] := 2.0;
   DATA[1646,25] := 2.0;
   DATA[1646,26] := 7.876058;
   DATA[1646,27] := 142.9121;
   DATA[1646,28] := 262.7852;
   DATA[1646,29] := 12.03538;
   DATA[1646,30] := 1.721738;
   DATA[1646,31] := 1.276162;
   DATA[1646,32] := 0.7355248;
   DATA[1646,33] := 0.3082983;
   DATA[1646,34] := 2.0;
   DATA[1646,35] := 249.984;
   DATA[1646,36] := 1.537821;
   DATA[1646,37] := 188.9259;
   DATA[1646,38] := 0.000128152;
   DATA[1646,39] := 1.0;
   DATA[1647,1] := 814.6125;
   DATA[1647,2] := 1.0;
   DATA[1647,3] := 1.0;
   DATA[1647,4] := 262.7211;
   DATA[1647,5] := 8.466932;
   DATA[1647,6] := 319.4053;
   DATA[1647,8] := 1.0;
   DATA[1647,9] := 1.0;
   DATA[1647,10] := 1.0;
   DATA[1647,11] := 19.74198;
   DATA[1647,12] := 2.213624;
   DATA[1647,13] := 878.701;
   DATA[1647,14] := 1.0;
   DATA[1647,15] := 2.0;
   DATA[1647,16] := 1.0;
   DATA[1647,17] := 1.0;
   DATA[1647,18] := 1.0;
   DATA[1647,19] := 2.0;
   DATA[1647,20] := 148.808;
   DATA[1647,21] := 154.1656;
   DATA[1647,22] := 1.717746;
   DATA[1647,23] := 799.5642;
   DATA[1647,24] := 2.0;
   DATA[1647,25] := 2.0;
   DATA[1647,26] := 7.876058;
   DATA[1647,27] := 142.9121;
   DATA[1647,28] := 262.7852;
   DATA[1647,29] := 12.03538;
   DATA[1647,30] := 1.721738;
   DATA[1647,31] := 1.291789;
   DATA[1647,32] := 0.7355248;
   DATA[1647,33] := 0.3082983;
   DATA[1647,34] := 2.0;
   DATA[1647,35] := 249.984;
   DATA[1647,36] := 1.762086;
   DATA[1647,37] := 188.9259;
   DATA[1647,38] := 0.000128152;
   DATA[1647,39] := 1.0;
   DATA[1648,1] := 814.534;
   DATA[1648,2] := 1.0;
   DATA[1648,3] := 1.0;
   DATA[1648,4] := 262.7211;
   DATA[1648,5] := 8.466932;
   DATA[1648,6] := 319.4053;
   DATA[1648,8] := 1.0;
   DATA[1648,9] := 1.0;
   DATA[1648,10] := 1.0;
   DATA[1648,11] := 19.75479;
   DATA[1648,12] := 2.213624;
   DATA[1648,13] := 878.1002;
   DATA[1648,14] := 1.0;
   DATA[1648,15] := 2.0;
   DATA[1648,16] := 1.0;
   DATA[1648,17] := 1.0;
   DATA[1648,18] := 1.0;
   DATA[1648,19] := 2.0;
   DATA[1648,20] := 148.808;
   DATA[1648,21] := 154.1656;
   DATA[1648,22] := 1.717746;
   DATA[1648,23] := 799.4104;
   DATA[1648,24] := 2.0;
   DATA[1648,25] := 2.0;
   DATA[1648,26] := 7.876058;
   DATA[1648,27] := 142.9121;
   DATA[1648,28] := 262.7852;
   DATA[1648,29] := 12.03538;
   DATA[1648,30] := 1.721738;
   DATA[1648,31] := 1.291918;
   DATA[1648,32] := 0.7355248;
   DATA[1648,33] := 0.3082983;
   DATA[1648,34] := 2.0;
   DATA[1648,35] := 249.984;
   DATA[1648,36] := 1.762086;
   DATA[1648,37] := 188.9259;
   DATA[1648,38] := 0.000128152;
   DATA[1648,39] := 1.0;
   DATA[1649,1] := 814.8088;
   DATA[1649,2] := 1.0;
   DATA[1649,3] := 1.0;
   DATA[1649,4] := 262.7211;
   DATA[1649,5] := 8.46533;
   DATA[1649,6] := 319.4053;
   DATA[1649,8] := 1.0;
   DATA[1649,9] := 1.0;
   DATA[1649,10] := 1.0;
   DATA[1649,11] := 19.7804;
   DATA[1649,12] := 2.212856;
   DATA[1649,13] := 877.98;
   DATA[1649,14] := 1.0;
   DATA[1649,15] := 2.0;
   DATA[1649,16] := 1.0;
   DATA[1649,17] := 1.0;
   DATA[1649,18] := 1.0;
   DATA[1649,19] := 2.0;
   DATA[1649,20] := 148.808;
   DATA[1649,21] := 154.1656;
   DATA[1649,22] := 1.71608;
   DATA[1649,23] := 799.6411;
   DATA[1649,24] := 2.0;
   DATA[1649,25] := 2.0;
   DATA[1649,26] := 7.876058;
   DATA[1649,27] := 142.9121;
   DATA[1649,28] := 262.7852;
   DATA[1649,29] := 12.03538;
   DATA[1649,30] := 1.723148;
   DATA[1649,31] := 1.30114;
   DATA[1649,32] := 0.7355248;
   DATA[1649,33] := 0.3082983;
   DATA[1649,34] := 2.0;
   DATA[1649,35] := 249.984;
   DATA[1649,36] := 1.69801;
   DATA[1649,37] := 188.8779;
   DATA[1649,38] := 0.000128152;
   DATA[1649,39] := 1.0;
   DATA[1650,1] := 815.1228;
   DATA[1650,2] := 1.0;
   DATA[1650,3] := 1.0;
   DATA[1650,4] := 262.5609;
   DATA[1650,5] := 8.46533;
   DATA[1650,6] := 319.4053;
   DATA[1650,8] := 1.0;
   DATA[1650,9] := 1.0;
   DATA[1650,10] := 1.0;
   DATA[1650,11] := 19.7804;
   DATA[1650,12] := 2.2126;
   DATA[1650,13] := 877.2991;
   DATA[1650,14] := 1.0;
   DATA[1650,15] := 2.0;
   DATA[1650,16] := 1.0;
   DATA[1650,17] := 1.0;
   DATA[1650,18] := 1.0;
   DATA[1650,19] := 2.0;
   DATA[1650,20] := 148.808;
   DATA[1650,21] := 154.1656;
   DATA[1650,22] := 1.71608;
   DATA[1650,23] := 799.5258;
   DATA[1650,24] := 2.0;
   DATA[1650,25] := 2.0;
   DATA[1650,26] := 7.876058;
   DATA[1650,27] := 142.9121;
   DATA[1650,28] := 262.7852;
   DATA[1650,29] := 12.03538;
   DATA[1650,30] := 1.724301;
   DATA[1650,31] := 1.302933;
   DATA[1650,32] := 0.7355248;
   DATA[1650,33] := 0.3082983;
   DATA[1650,34] := 2.0;
   DATA[1650,35] := 249.984;
   DATA[1650,36] := 1.617916;
   DATA[1650,37] := 188.8779;
   DATA[1650,38] := 0.000128152;
   DATA[1650,39] := 1.0;
   DATA[1651,1] := 815.0835;
   DATA[1651,2] := 1.0;
   DATA[1651,3] := 1.0;
   DATA[1651,4] := 262.5609;
   DATA[1651,5] := 8.46533;
   DATA[1651,6] := 319.4053;
   DATA[1651,8] := 1.0;
   DATA[1651,9] := 1.0;
   DATA[1651,10] := 1.0;
   DATA[1651,11] := 19.7804;
   DATA[1651,12] := 2.2126;
   DATA[1651,13] := 876.9386;
   DATA[1651,14] := 1.0;
   DATA[1651,15] := 2.0;
   DATA[1651,16] := 1.0;
   DATA[1651,17] := 1.0;
   DATA[1651,18] := 1.0;
   DATA[1651,19] := 2.0;
   DATA[1651,20] := 148.808;
   DATA[1651,21] := 154.1656;
   DATA[1651,22] := 1.71608;
   DATA[1651,23] := 799.1412;
   DATA[1651,24] := 2.0;
   DATA[1651,25] := 2.0;
   DATA[1651,26] := 7.876058;
   DATA[1651,27] := 142.9121;
   DATA[1651,28] := 262.7852;
   DATA[1651,29] := 12.03538;
   DATA[1651,30] := 1.724301;
   DATA[1651,31] := 1.298578;
   DATA[1651,32] := 0.7355248;
   DATA[1651,33] := 0.3082983;
   DATA[1651,34] := 2.0;
   DATA[1651,35] := 249.984;
   DATA[1651,36] := 1.617916;
   DATA[1651,37] := 188.8779;
   DATA[1651,38] := 0.000128152;
   DATA[1651,39] := 1.0;
   DATA[1652,1] := 814.9658;
   DATA[1652,2] := 1.0;
   DATA[1652,3] := 1.0;
   DATA[1652,4] := 262.5609;
   DATA[1652,5] := 8.46533;
   DATA[1652,6] := 319.4053;
   DATA[1652,8] := 1.0;
   DATA[1652,9] := 1.0;
   DATA[1652,10] := 1.0;
   DATA[1652,11] := 19.7804;
   DATA[1652,12] := 2.2126;
   DATA[1652,13] := 876.2177;
   DATA[1652,14] := 1.0;
   DATA[1652,15] := 2.0;
   DATA[1652,16] := 1.0;
   DATA[1652,17] := 1.0;
   DATA[1652,18] := 1.0;
   DATA[1652,19] := 2.0;
   DATA[1652,20] := 148.808;
   DATA[1652,21] := 154.0118;
   DATA[1652,22] := 1.714286;
   DATA[1652,23] := 799.4104;
   DATA[1652,24] := 2.0;
   DATA[1652,25] := 2.0;
   DATA[1652,26] := 7.876058;
   DATA[1652,27] := 142.9121;
   DATA[1652,28] := 262.7852;
   DATA[1652,29] := 12.03538;
   DATA[1652,30] := 1.724301;
   DATA[1652,31] := 1.291918;
   DATA[1652,32] := 0.7355248;
   DATA[1652,33] := 0.3082983;
   DATA[1652,34] := 2.0;
   DATA[1652,35] := 249.984;
   DATA[1652,36] := 1.617916;
   DATA[1652,37] := 188.8779;
   DATA[1652,38] := 0.000128152;
   DATA[1652,39] := 1.0;
   DATA[1653,1] := 814.8873;
   DATA[1653,2] := 1.0;
   DATA[1653,3] := 1.0;
   DATA[1653,4] := 262.5609;
   DATA[1653,5] := 8.46533;
   DATA[1653,6] := 319.4053;
   DATA[1653,8] := 1.0;
   DATA[1653,9] := 1.0;
   DATA[1653,10] := 1.0;
   DATA[1653,11] := 19.72598;
   DATA[1653,12] := 2.2126;
   DATA[1653,13] := 875.737;
   DATA[1653,14] := 1.0;
   DATA[1653,15] := 2.0;
   DATA[1653,16] := 1.0;
   DATA[1653,17] := 1.0;
   DATA[1653,18] := 1.0;
   DATA[1653,19] := 2.0;
   DATA[1653,20] := 148.808;
   DATA[1653,21] := 154.0118;
   DATA[1653,22] := 1.713517;
   DATA[1653,23] := 799.4104;
   DATA[1653,24] := 2.0;
   DATA[1653,25] := 2.0;
   DATA[1653,26] := 7.876058;
   DATA[1653,27] := 142.9121;
   DATA[1653,28] := 262.7852;
   DATA[1653,29] := 12.30454;
   DATA[1653,30] := 1.724301;
   DATA[1653,31] := 1.299731;
   DATA[1653,32] := 0.7355248;
   DATA[1653,33] := 0.3082983;
   DATA[1653,34] := 2.0;
   DATA[1653,35] := 249.984;
   DATA[1653,36] := 1.617916;
   DATA[1653,37] := 188.8779;
   DATA[1653,38] := 0.000128152;
   DATA[1653,39] := 1.0;
   DATA[1654,1] := 815.0835;
   DATA[1654,2] := 1.0;
   DATA[1654,3] := 1.0;
   DATA[1654,4] := 262.5609;
   DATA[1654,5] := 8.46533;
   DATA[1654,6] := 319.4053;
   DATA[1654,8] := 1.0;
   DATA[1654,9] := 1.0;
   DATA[1654,10] := 1.0;
   DATA[1654,11] := 19.72598;
   DATA[1654,12] := 2.2126;
   DATA[1654,13] := 875.1763;
   DATA[1654,14] := 1.0;
   DATA[1654,15] := 2.0;
   DATA[1654,16] := 1.0;
   DATA[1654,17] := 1.0;
   DATA[1654,18] := 1.0;
   DATA[1654,19] := 2.0;
   DATA[1654,20] := 148.808;
   DATA[1654,21] := 153.9862;
   DATA[1654,22] := 1.713389;
   DATA[1654,23] := 799.2181;
   DATA[1654,24] := 2.0;
   DATA[1654,25] := 2.0;
   DATA[1654,26] := 7.876058;
   DATA[1654,27] := 142.9121;
   DATA[1654,28] := 262.7852;
   DATA[1654,29] := 12.30454;
   DATA[1654,30] := 1.724301;
   DATA[1654,31] := 1.296529;
   DATA[1654,32] := 0.7355248;
   DATA[1654,33] := 0.3082983;
   DATA[1654,34] := 2.0;
   DATA[1654,35] := 249.984;
   DATA[1654,36] := 1.617916;
   DATA[1654,37] := 188.8779;
   DATA[1654,38] := 0.000128152;
   DATA[1654,39] := 1.0;
   DATA[1655,1] := 815.2798;
   DATA[1655,2] := 1.0;
   DATA[1655,3] := 1.0;
   DATA[1655,4] := 262.5609;
   DATA[1655,5] := 8.46533;
   DATA[1655,6] := 319.4053;
   DATA[1655,8] := 1.0;
   DATA[1655,9] := 1.0;
   DATA[1655,10] := 1.0;
   DATA[1655,11] := 19.72598;
   DATA[1655,12] := 2.211831;
   DATA[1655,13] := 874.6155;
   DATA[1655,14] := 1.0;
   DATA[1655,15] := 2.0;
   DATA[1655,16] := 1.0;
   DATA[1655,17] := 1.0;
   DATA[1655,18] := 1.0;
   DATA[1655,19] := 2.0;
   DATA[1655,20] := 148.808;
   DATA[1655,21] := 153.9862;
   DATA[1655,22] := 1.713389;
   DATA[1655,23] := 799.1412;
   DATA[1655,24] := 2.0;
   DATA[1655,25] := 2.0;
   DATA[1655,26] := 7.876058;
   DATA[1655,27] := 142.9121;
   DATA[1655,28] := 262.7852;
   DATA[1655,29] := 12.30454;
   DATA[1655,30] := 1.724301;
   DATA[1655,31] := 1.297169;
   DATA[1655,32] := 0.7355248;
   DATA[1655,33] := 0.3082983;
   DATA[1655,34] := 2.0;
   DATA[1655,35] := 249.984;
   DATA[1655,36] := 1.617916;
   DATA[1655,37] := 188.8779;
   DATA[1655,38] := 0.000128152;
   DATA[1655,39] := 1.0;
   DATA[1656,1] := 815.3583;
   DATA[1656,2] := 1.0;
   DATA[1656,3] := 1.0;
   DATA[1656,4] := 262.5609;
   DATA[1656,5] := 8.46533;
   DATA[1656,6] := 319.4053;
   DATA[1656,8] := 1.0;
   DATA[1656,9] := 1.0;
   DATA[1656,10] := 1.0;
   DATA[1656,11] := 19.72598;
   DATA[1656,12] := 2.209397;
   DATA[1656,13] := 874.4954;
   DATA[1656,14] := 1.0;
   DATA[1656,15] := 2.0;
   DATA[1656,16] := 1.0;
   DATA[1656,17] := 1.0;
   DATA[1656,18] := 1.0;
   DATA[1656,19] := 2.0;
   DATA[1656,20] := 148.808;
   DATA[1656,21] := 153.9862;
   DATA[1656,22] := 1.711595;
   DATA[1656,23] := 799.5642;
   DATA[1656,24] := 2.0;
   DATA[1656,25] := 2.0;
   DATA[1656,26] := 7.876058;
   DATA[1656,27] := 143.0403;
   DATA[1656,28] := 262.7852;
   DATA[1656,29] := 12.26609;
   DATA[1656,30] := 1.724301;
   DATA[1656,31] := 1.291149;
   DATA[1656,32] := 0.7355248;
   DATA[1656,33] := 0.3082983;
   DATA[1656,34] := 2.0;
   DATA[1656,35] := 249.984;
   DATA[1656,36] := 1.617916;
   DATA[1656,37] := 188.8779;
   DATA[1656,38] := 0.000128152;
   DATA[1656,39] := 1.0;
   DATA[1657,1] := 815.3583;
   DATA[1657,2] := 1.0;
   DATA[1657,3] := 1.0;
   DATA[1657,4] := 262.5609;
   DATA[1657,5] := 8.46533;
   DATA[1657,6] := 319.4053;
   DATA[1657,8] := 1.0;
   DATA[1657,9] := 1.0;
   DATA[1657,10] := 1.0;
   DATA[1657,11] := 19.72598;
   DATA[1657,12] := 2.209397;
   DATA[1657,13] := 873.7744;
   DATA[1657,14] := 1.0;
   DATA[1657,15] := 2.0;
   DATA[1657,16] := 1.0;
   DATA[1657,17] := 1.0;
   DATA[1657,18] := 1.0;
   DATA[1657,19] := 2.0;
   DATA[1657,20] := 148.808;
   DATA[1657,21] := 153.9862;
   DATA[1657,22] := 1.711595;
   DATA[1657,23] := 800.0256;
   DATA[1657,24] := 2.0;
   DATA[1657,25] := 2.0;
   DATA[1657,26] := 7.876058;
   DATA[1657,27] := 143.0403;
   DATA[1657,28] := 262.7852;
   DATA[1657,29] := 12.15073;
   DATA[1657,30] := 1.722379;
   DATA[1657,31] := 1.268093;
   DATA[1657,32] := 0.7355248;
   DATA[1657,33] := 0.3082983;
   DATA[1657,34] := 2.0;
   DATA[1657,35] := 249.984;
   DATA[1657,36] := 1.617916;
   DATA[1657,37] := 188.8779;
   DATA[1657,38] := 0.000128152;
   DATA[1657,39] := 1.0;
   DATA[1658,1] := 815.3583;
   DATA[1658,2] := 1.0;
   DATA[1658,3] := 1.0;
   DATA[1658,4] := 262.5609;
   DATA[1658,5] := 8.46533;
   DATA[1658,6] := 319.4053;
   DATA[1658,8] := 1.0;
   DATA[1658,9] := 1.0;
   DATA[1658,10] := 1.0;
   DATA[1658,11] := 19.72598;
   DATA[1658,12] := 2.212087;
   DATA[1658,13] := 873.1736;
   DATA[1658,14] := 1.0;
   DATA[1658,15] := 2.0;
   DATA[1658,16] := 1.0;
   DATA[1658,17] := 1.0;
   DATA[1658,18] := 1.0;
   DATA[1658,19] := 2.0;
   DATA[1658,20] := 148.808;
   DATA[1658,21] := 153.9862;
   DATA[1658,22] := 1.711595;
   DATA[1658,23] := 799.7949;
   DATA[1658,24] := 2.0;
   DATA[1658,25] := 2.0;
   DATA[1658,26] := 7.876058;
   DATA[1658,27] := 143.0403;
   DATA[1658,28] := 262.7852;
   DATA[1658,29] := 12.15073;
   DATA[1658,30] := 1.722379;
   DATA[1658,31] := 1.248111;
   DATA[1658,32] := 0.7355248;
   DATA[1658,33] := 0.3082983;
   DATA[1658,34] := 2.0;
   DATA[1658,35] := 249.984;
   DATA[1658,36] := 1.617916;
   DATA[1658,37] := 188.7016;
   DATA[1658,38] := 0.000128152;
   DATA[1658,39] := 1.0;
   DATA[1659,1] := 815.5153;
   DATA[1659,2] := 1.0;
   DATA[1659,3] := 1.0;
   DATA[1659,4] := 262.5609;
   DATA[1659,5] := 8.46533;
   DATA[1659,6] := 319.4053;
   DATA[1659,8] := 1.0;
   DATA[1659,9] := 1.0;
   DATA[1659,10] := 1.0;
   DATA[1659,11] := 19.7836;
   DATA[1659,12] := 2.212087;
   DATA[1659,13] := 872.733;
   DATA[1659,14] := 1.0;
   DATA[1659,15] := 2.0;
   DATA[1659,16] := 1.0;
   DATA[1659,17] := 1.0;
   DATA[1659,18] := 1.0;
   DATA[1659,19] := 2.0;
   DATA[1659,20] := 148.808;
   DATA[1659,21] := 153.9862;
   DATA[1659,22] := 1.711595;
   DATA[1659,23] := 799.5642;
   DATA[1659,24] := 2.0;
   DATA[1659,25] := 2.0;
   DATA[1659,26] := 7.876058;
   DATA[1659,27] := 143.0403;
   DATA[1659,28] := 262.7852;
   DATA[1659,29] := 12.15073;
   DATA[1659,30] := 1.722379;
   DATA[1659,31] := 1.235942;
   DATA[1659,32] := 0.7355248;
   DATA[1659,33] := 0.3082983;
   DATA[1659,34] := 2.0;
   DATA[1659,35] := 249.8238;
   DATA[1659,36] := 1.617916;
   DATA[1659,37] := 188.7016;
   DATA[1659,38] := 0.000128152;
   DATA[1659,39] := 1.0;
   DATA[1660,1] := 815.3583;
   DATA[1660,2] := 1.0;
   DATA[1660,3] := 1.0;
   DATA[1660,4] := 262.5609;
   DATA[1660,5] := 8.46533;
   DATA[1660,6] := 319.4053;
   DATA[1660,8] := 1.0;
   DATA[1660,9] := 1.0;
   DATA[1660,10] := 1.0;
   DATA[1660,11] := 19.7836;
   DATA[1660,12] := 2.210934;
   DATA[1660,13] := 872.3725;
   DATA[1660,14] := 1.0;
   DATA[1660,15] := 2.0;
   DATA[1660,16] := 1.0;
   DATA[1660,17] := 1.0;
   DATA[1660,18] := 1.0;
   DATA[1660,19] := 2.0;
   DATA[1660,20] := 148.808;
   DATA[1660,21] := 153.9862;
   DATA[1660,22] := 1.711595;
   DATA[1660,23] := 799.9487;
   DATA[1660,24] := 2.0;
   DATA[1660,25] := 2.0;
   DATA[1660,26] := 7.876058;
   DATA[1660,27] := 143.0403;
   DATA[1660,28] := 262.6891;
   DATA[1660,29] := 12.15073;
   DATA[1660,30] := 1.722379;
   DATA[1660,31] := 1.243115;
   DATA[1660,32] := 0.7355248;
   DATA[1660,33] := 0.3082983;
   DATA[1660,34] := 2.0;
   DATA[1660,35] := 249.8238;
   DATA[1660,36] := 1.617916;
   DATA[1660,37] := 188.6375;
   DATA[1660,38] := 0.000128152;
   DATA[1660,39] := 1.0;
   DATA[1661,1] := 815.162;
   DATA[1661,2] := 1.0;
   DATA[1661,3] := 1.0;
   DATA[1661,4] := 262.5609;
   DATA[1661,5] := 8.46533;
   DATA[1661,6] := 319.4053;
   DATA[1661,8] := 1.0;
   DATA[1661,9] := 1.0;
   DATA[1661,10] := 1.0;
   DATA[1661,11] := 19.7836;
   DATA[1661,12] := 2.209653;
   DATA[1661,13] := 871.5314;
   DATA[1661,14] := 1.0;
   DATA[1661,15] := 2.0;
   DATA[1661,16] := 1.0;
   DATA[1661,17] := 1.0;
   DATA[1661,18] := 1.0;
   DATA[1661,19] := 2.0;
   DATA[1661,20] := 148.808;
   DATA[1661,21] := 153.9862;
   DATA[1661,22] := 1.711595;
   DATA[1661,23] := 799.6411;
   DATA[1661,24] := 2.0;
   DATA[1661,25] := 2.0;
   DATA[1661,26] := 7.876058;
   DATA[1661,27] := 143.0403;
   DATA[1661,28] := 262.6891;
   DATA[1661,29] := 12.15073;
   DATA[1661,30] := 1.722379;
   DATA[1661,31] := 1.263994;
   DATA[1661,32] := 0.7355248;
   DATA[1661,33] := 0.3082983;
   DATA[1661,34] := 2.0;
   DATA[1661,35] := 249.8238;
   DATA[1661,36] := 1.617916;
   DATA[1661,37] := 188.6375;
   DATA[1661,38] := 0.000128152;
   DATA[1661,39] := 1.0;
   DATA[1662,1] := 815.005;
   DATA[1662,2] := 1.0;
   DATA[1662,3] := 1.0;
   DATA[1662,4] := 262.5609;
   DATA[1662,5] := 8.46533;
   DATA[1662,6] := 319.4053;
   DATA[1662,8] := 1.0;
   DATA[1662,9] := 1.0;
   DATA[1662,10] := 1.0;
   DATA[1662,11] := 19.7836;
   DATA[1662,12] := 2.209653;
   DATA[1662,13] := 871.291;
   DATA[1662,14] := 1.0;
   DATA[1662,15] := 2.0;
   DATA[1662,16] := 1.0;
   DATA[1662,17] := 1.0;
   DATA[1662,18] := 1.0;
   DATA[1662,19] := 2.0;
   DATA[1662,20] := 148.808;
   DATA[1662,21] := 153.9862;
   DATA[1662,22] := 1.710313;
   DATA[1662,23] := 799.7949;
   DATA[1662,24] := 2.0;
   DATA[1662,25] := 2.0;
   DATA[1662,26] := 7.876058;
   DATA[1662,27] := 143.0403;
   DATA[1662,28] := 262.6891;
   DATA[1662,29] := 12.15073;
   DATA[1662,30] := 1.724686;
   DATA[1662,31] := 1.271423;
   DATA[1662,32] := 0.7355248;
   DATA[1662,33] := 0.3082983;
   DATA[1662,34] := 2.0;
   DATA[1662,35] := 249.8238;
   DATA[1662,36] := 1.617916;
   DATA[1662,37] := 188.6375;
   DATA[1662,38] := 0.000128152;
   DATA[1662,39] := 1.0;
   DATA[1663,1] := 815.005;
   DATA[1663,2] := 1.0;
   DATA[1663,3] := 1.0;
   DATA[1663,4] := 262.5609;
   DATA[1663,5] := 8.46533;
   DATA[1663,6] := 319.4053;
   DATA[1663,8] := 1.0;
   DATA[1663,9] := 1.0;
   DATA[1663,10] := 1.0;
   DATA[1663,11] := 19.85402;
   DATA[1663,12] := 2.209653;
   DATA[1663,13] := 870.6101;
   DATA[1663,14] := 1.0;
   DATA[1663,15] := 2.0;
   DATA[1663,16] := 1.0;
   DATA[1663,17] := 1.0;
   DATA[1663,18] := 1.0;
   DATA[1663,19] := 2.0;
   DATA[1663,20] := 148.808;
   DATA[1663,21] := 153.9862;
   DATA[1663,22] := 1.710313;
   DATA[1663,23] := 799.5258;
   DATA[1663,24] := 2.0;
   DATA[1663,25] := 2.0;
   DATA[1663,26] := 7.876058;
   DATA[1663,27] := 143.0403;
   DATA[1663,28] := 262.6891;
   DATA[1663,29] := 12.15073;
   DATA[1663,30] := 1.724686;
   DATA[1663,31] := 1.272064;
   DATA[1663,32] := 0.7355248;
   DATA[1663,33] := 0.3082983;
   DATA[1663,34] := 2.0;
   DATA[1663,35] := 249.8238;
   DATA[1663,36] := 1.617916;
   DATA[1663,37] := 188.6375;
   DATA[1663,38] := 0.000128152;
   DATA[1663,39] := 1.0;
   DATA[1664,1] := 815.3583;
   DATA[1664,2] := 1.0;
   DATA[1664,3] := 1.0;
   DATA[1664,4] := 262.5609;
   DATA[1664,5] := 8.46533;
   DATA[1664,6] := 319.4053;
   DATA[1664,8] := 1.0;
   DATA[1664,9] := 1.0;
   DATA[1664,10] := 1.0;
   DATA[1664,11] := 19.87003;
   DATA[1664,12] := 2.209653;
   DATA[1664,13] := 870.7303;
   DATA[1664,14] := 1.0;
   DATA[1664,15] := 2.0;
   DATA[1664,16] := 1.0;
   DATA[1664,17] := 1.0;
   DATA[1664,18] := 1.0;
   DATA[1664,19] := 2.0;
   DATA[1664,20] := 148.808;
   DATA[1664,21] := 153.9862;
   DATA[1664,22] := 1.713389;
   DATA[1664,23] := 799.5258;
   DATA[1664,24] := 2.0;
   DATA[1664,25] := 2.0;
   DATA[1664,26] := 7.876058;
   DATA[1664,27] := 143.0403;
   DATA[1664,28] := 262.6891;
   DATA[1664,29] := 12.15073;
   DATA[1664,30] := 1.724686;
   DATA[1664,31] := 1.282183;
   DATA[1664,32] := 0.7355248;
   DATA[1664,33] := 0.3082983;
   DATA[1664,34] := 2.0;
   DATA[1664,35] := 249.8238;
   DATA[1664,36] := 1.617916;
   DATA[1664,37] := 188.7176;
   DATA[1664,38] := 0.000128152;
   DATA[1664,39] := 1.0;
   DATA[1665,1] := 815.319;
   DATA[1665,2] := 1.0;
   DATA[1665,3] := 1.0;
   DATA[1665,4] := 262.5609;
   DATA[1665,5] := 8.46533;
   DATA[1665,6] := 319.4053;
   DATA[1665,8] := 1.0;
   DATA[1665,9] := 1.0;
   DATA[1665,10] := 1.0;
   DATA[1665,11] := 19.87003;
   DATA[1665,12] := 2.209653;
   DATA[1665,13] := 869.8892;
   DATA[1665,14] := 1.0;
   DATA[1665,15] := 2.0;
   DATA[1665,16] := 1.0;
   DATA[1665,17] := 1.0;
   DATA[1665,18] := 1.0;
   DATA[1665,19] := 2.0;
   DATA[1665,20] := 148.808;
   DATA[1665,21] := 153.9862;
   DATA[1665,22] := 1.713389;
   DATA[1665,23] := 799.8334;
   DATA[1665,24] := 2.0;
   DATA[1665,25] := 2.0;
   DATA[1665,26] := 7.876058;
   DATA[1665,27] := 143.0403;
   DATA[1665,28] := 262.6891;
   DATA[1665,29] := 12.15073;
   DATA[1665,30] := 1.724686;
   DATA[1665,31] := 1.292814;
   DATA[1665,32] := 0.7355248;
   DATA[1665,33] := 0.3082983;
   DATA[1665,34] := 2.0;
   DATA[1665,35] := 250.0;
   DATA[1665,36] := 1.617916;
   DATA[1665,37] := 188.8779;
   DATA[1665,38] := 0.000128152;
   DATA[1665,39] := 1.0;
   DATA[1666,1] := 815.2798;
   DATA[1666,2] := 1.0;
   DATA[1666,3] := 1.0;
   DATA[1666,4] := 262.657;
   DATA[1666,5] := 8.46533;
   DATA[1666,6] := 319.4053;
   DATA[1666,8] := 1.0;
   DATA[1666,9] := 1.0;
   DATA[1666,10] := 1.0;
   DATA[1666,11] := 19.87003;
   DATA[1666,12] := 2.209653;
   DATA[1666,13] := 869.3284;
   DATA[1666,14] := 1.0;
   DATA[1666,15] := 2.0;
   DATA[1666,16] := 1.0;
   DATA[1666,17] := 1.0;
   DATA[1666,18] := 1.0;
   DATA[1666,19] := 2.0;
   DATA[1666,20] := 148.808;
   DATA[1666,21] := 153.9862;
   DATA[1666,22] := 1.713389;
   DATA[1666,23] := 800.0256;
   DATA[1666,24] := 2.0;
   DATA[1666,25] := 2.0;
   DATA[1666,26] := 7.876058;
   DATA[1666,27] := 143.0403;
   DATA[1666,28] := 262.6891;
   DATA[1666,29] := 12.15073;
   DATA[1666,30] := 1.724045;
   DATA[1666,31] := 1.303574;
   DATA[1666,32] := 0.7355248;
   DATA[1666,33] := 0.3082983;
   DATA[1666,34] := 2.0;
   DATA[1666,35] := 250.0;
   DATA[1666,36] := 1.617916;
   DATA[1666,37] := 188.8779;
   DATA[1666,38] := 0.000128152;
   DATA[1666,39] := 1.0;
   DATA[1667,1] := 815.4761;
   DATA[1667,2] := 1.0;
   DATA[1667,3] := 1.0;
   DATA[1667,4] := 262.657;
   DATA[1667,5] := 8.46533;
   DATA[1667,6] := 319.4053;
   DATA[1667,8] := 1.0;
   DATA[1667,9] := 1.0;
   DATA[1667,10] := 1.0;
   DATA[1667,11] := 19.87003;
   DATA[1667,12] := 2.209653;
   DATA[1667,13] := 868.5273;
   DATA[1667,14] := 1.0;
   DATA[1667,15] := 2.0;
   DATA[1667,16] := 1.0;
   DATA[1667,17] := 1.0;
   DATA[1667,18] := 1.0;
   DATA[1667,19] := 2.0;
   DATA[1667,20] := 148.808;
   DATA[1667,21] := 153.9862;
   DATA[1667,22] := 1.715183;
   DATA[1667,23] := 799.7949;
   DATA[1667,24] := 2.0;
   DATA[1667,25] := 2.0;
   DATA[1667,26] := 7.876058;
   DATA[1667,27] := 142.989;
   DATA[1667,28] := 262.6891;
   DATA[1667,29] := 12.15073;
   DATA[1667,30] := 1.724045;
   DATA[1667,31] := 1.311259;
   DATA[1667,32] := 0.7355248;
   DATA[1667,33] := 0.3082983;
   DATA[1667,34] := 2.0;
   DATA[1667,35] := 250.0;
   DATA[1667,36] := 1.617916;
   DATA[1667,37] := 188.8779;
   DATA[1667,38] := 0.000128152;
   DATA[1667,39] := 1.0;
   DATA[1668,1] := 815.5938;
   DATA[1668,2] := 1.0;
   DATA[1668,3] := 1.0;
   DATA[1668,4] := 262.657;
   DATA[1668,5] := 8.46533;
   DATA[1668,6] := 319.4053;
   DATA[1668,8] := 1.0;
   DATA[1668,9] := 1.0;
   DATA[1668,10] := 1.0;
   DATA[1668,11] := 19.75159;
   DATA[1668,12] := 2.209653;
   DATA[1668,13] := 868.5273;
   DATA[1668,14] := 1.0;
   DATA[1668,15] := 2.0;
   DATA[1668,16] := 1.0;
   DATA[1668,17] := 1.0;
   DATA[1668,18] := 1.0;
   DATA[1668,19] := 2.0;
   DATA[1668,20] := 148.808;
   DATA[1668,21] := 153.9862;
   DATA[1668,22] := 1.71608;
   DATA[1668,23] := 800.1025;
   DATA[1668,24] := 2.0;
   DATA[1668,25] := 2.0;
   DATA[1668,26] := 7.876058;
   DATA[1668,27] := 142.989;
   DATA[1668,28] := 262.6891;
   DATA[1668,29] := 12.15073;
   DATA[1668,30] := 1.724045;
   DATA[1668,31] := 1.305495;
   DATA[1668,32] := 0.7355248;
   DATA[1668,33] := 0.3082983;
   DATA[1668,34] := 2.0;
   DATA[1668,35] := 250.0;
   DATA[1668,36] := 1.617916;
   DATA[1668,37] := 188.8779;
   DATA[1668,38] := 0.000128152;
   DATA[1668,39] := 1.0;
   DATA[1669,1] := 815.4761;
   DATA[1669,2] := 1.0;
   DATA[1669,3] := 1.0;
   DATA[1669,4] := 262.657;
   DATA[1669,5] := 8.46533;
   DATA[1669,6] := 319.4053;
   DATA[1669,8] := 1.0;
   DATA[1669,9] := 1.0;
   DATA[1669,10] := 1.0;
   DATA[1669,11] := 19.75159;
   DATA[1669,12] := 2.209653;
   DATA[1669,13] := 867.9265;
   DATA[1669,14] := 1.0;
   DATA[1669,15] := 2.0;
   DATA[1669,16] := 1.0;
   DATA[1669,17] := 1.0;
   DATA[1669,18] := 1.0;
   DATA[1669,19] := 2.0;
   DATA[1669,20] := 148.808;
   DATA[1669,21] := 153.9862;
   DATA[1669,22] := 1.71608;
   DATA[1669,23] := 800.2179;
   DATA[1669,24] := 2.0;
   DATA[1669,25] := 2.0;
   DATA[1669,26] := 7.876058;
   DATA[1669,27] := 142.989;
   DATA[1669,28] := 262.6891;
   DATA[1669,29] := 12.15073;
   DATA[1669,30] := 1.722892;
   DATA[1669,31] := 1.30114;
   DATA[1669,32] := 0.7355248;
   DATA[1669,33] := 0.3082983;
   DATA[1669,34] := 2.0;
   DATA[1669,35] := 250.0;
   DATA[1669,36] := 1.69801;
   DATA[1669,37] := 188.8779;
   DATA[1669,38] := 0.000128152;
   DATA[1669,39] := 1.0;
   DATA[1670,1] := 815.4761;
   DATA[1670,2] := 1.0;
   DATA[1670,3] := 1.0;
   DATA[1670,4] := 262.657;
   DATA[1670,5] := 8.46533;
   DATA[1670,6] := 319.4053;
   DATA[1670,8] := 1.0;
   DATA[1670,9] := 1.0;
   DATA[1670,10] := 1.0;
   DATA[1670,11] := 19.75159;
   DATA[1670,12] := 2.209909;
   DATA[1670,13] := 867.7263;
   DATA[1670,14] := 1.0;
   DATA[1670,15] := 2.0;
   DATA[1670,16] := 1.0;
   DATA[1670,17] := 1.0;
   DATA[1670,18] := 1.0;
   DATA[1670,19] := 2.0;
   DATA[1670,20] := 148.808;
   DATA[1670,21] := 153.9862;
   DATA[1670,22] := 1.716592;
   DATA[1670,23] := 800.3333;
   DATA[1670,24] := 2.0;
   DATA[1670,25] := 2.0;
   DATA[1670,26] := 7.876058;
   DATA[1670,27] := 142.9377;
   DATA[1670,28] := 262.6891;
   DATA[1670,29] := 12.15073;
   DATA[1670,30] := 1.721866;
   DATA[1670,31] := 1.30114;
   DATA[1670,32] := 0.7355248;
   DATA[1670,33] := 0.3082983;
   DATA[1670,34] := 2.0;
   DATA[1670,35] := 250.0;
   DATA[1670,36] := 1.69801;
   DATA[1670,37] := 188.8779;
   DATA[1670,38] := 0.000128152;
   DATA[1670,39] := 1.0;
   DATA[1671,1] := 815.4761;
   DATA[1671,2] := 1.0;
   DATA[1671,3] := 1.0;
   DATA[1671,4] := 262.657;
   DATA[1671,5] := 8.46533;
   DATA[1671,6] := 319.4053;
   DATA[1671,8] := 1.0;
   DATA[1671,9] := 1.0;
   DATA[1671,10] := 1.0;
   DATA[1671,11] := 19.75159;
   DATA[1671,12] := 2.209909;
   DATA[1671,13] := 867.1655;
   DATA[1671,14] := 1.0;
   DATA[1671,15] := 2.0;
   DATA[1671,16] := 1.0;
   DATA[1671,17] := 1.0;
   DATA[1671,18] := 1.0;
   DATA[1671,19] := 2.0;
   DATA[1671,20] := 148.808;
   DATA[1671,21] := 153.9862;
   DATA[1671,22] := 1.716592;
   DATA[1671,23] := 800.5255;
   DATA[1671,24] := 2.0;
   DATA[1671,25] := 2.0;
   DATA[1671,26] := 7.876058;
   DATA[1671,27] := 142.9377;
   DATA[1671,28] := 262.6891;
   DATA[1671,29] := 12.15073;
   DATA[1671,30] := 1.721866;
   DATA[1671,31] := 1.290765;
   DATA[1671,32] := 0.7355248;
   DATA[1671,33] := 0.3082983;
   DATA[1671,34] := 2.0;
   DATA[1671,35] := 250.0;
   DATA[1671,36] := 1.69801;
   DATA[1671,37] := 188.8779;
   DATA[1671,38] := 0.000128152;
   DATA[1671,39] := 1.0;
   DATA[1672,1] := 815.319;
   DATA[1672,2] := 1.0;
   DATA[1672,3] := 1.0;
   DATA[1672,4] := 262.657;
   DATA[1672,5] := 8.46533;
   DATA[1672,6] := 319.4053;
   DATA[1672,8] := 1.0;
   DATA[1672,9] := 1.0;
   DATA[1672,10] := 1.0;
   DATA[1672,11] := 19.79;
   DATA[1672,12] := 2.211447;
   DATA[1672,13] := 866.9252;
   DATA[1672,14] := 1.0;
   DATA[1672,15] := 2.0;
   DATA[1672,16] := 1.0;
   DATA[1672,17] := 1.0;
   DATA[1672,18] := 1.0;
   DATA[1672,19] := 2.0;
   DATA[1672,20] := 148.808;
   DATA[1672,21] := 153.9862;
   DATA[1672,22] := 1.713261;
   DATA[1672,23] := 800.5255;
   DATA[1672,24] := 2.0;
   DATA[1672,25] := 2.0;
   DATA[1672,26] := 7.876058;
   DATA[1672,27] := 142.9377;
   DATA[1672,28] := 262.6891;
   DATA[1672,29] := 12.15073;
   DATA[1672,30] := 1.721866;
   DATA[1672,31] := 1.279749;
   DATA[1672,32] := 0.7355248;
   DATA[1672,33] := 0.3082983;
   DATA[1672,34] := 2.0;
   DATA[1672,35] := 250.0;
   DATA[1672,36] := 1.69801;
   DATA[1672,37] := 188.8138;
   DATA[1672,38] := 0.000128152;
   DATA[1672,39] := 1.0;
   DATA[1673,1] := 815.5153;
   DATA[1673,2] := 1.0;
   DATA[1673,3] := 1.0;
   DATA[1673,4] := 262.657;
   DATA[1673,5] := 8.46533;
   DATA[1673,6] := 319.4053;
   DATA[1673,8] := 1.0;
   DATA[1673,9] := 1.0;
   DATA[1673,10] := 1.0;
   DATA[1673,11] := 19.79;
   DATA[1673,12] := 2.211447;
   DATA[1673,13] := 866.7249;
   DATA[1673,14] := 1.0;
   DATA[1673,15] := 2.0;
   DATA[1673,16] := 1.0;
   DATA[1673,17] := 1.0;
   DATA[1673,18] := 1.0;
   DATA[1673,19] := 2.0;
   DATA[1673,20] := 148.808;
   DATA[1673,21] := 153.9862;
   DATA[1673,22] := 1.713261;
   DATA[1673,23] := 800.7562;
   DATA[1673,24] := 2.0;
   DATA[1673,25] := 2.0;
   DATA[1673,26] := 7.876058;
   DATA[1673,27] := 142.9377;
   DATA[1673,28] := 262.6891;
   DATA[1673,29] := 12.15073;
   DATA[1673,30] := 1.721866;
   DATA[1673,31] := 1.271679;
   DATA[1673,32] := 0.7355248;
   DATA[1673,33] := 0.3082983;
   DATA[1673,34] := 2.0;
   DATA[1673,35] := 249.8238;
   DATA[1673,36] := 1.585878;
   DATA[1673,37] := 188.7337;
   DATA[1673,38] := 0.000128152;
   DATA[1673,39] := 1.0;
   DATA[1674,1] := 815.3583;
   DATA[1674,2] := 1.0;
   DATA[1674,3] := 1.0;
   DATA[1674,4] := 262.657;
   DATA[1674,5] := 8.46533;
   DATA[1674,6] := 319.4053;
   DATA[1674,8] := 1.0;
   DATA[1674,9] := 1.0;
   DATA[1674,10] := 1.0;
   DATA[1674,11] := 19.79;
   DATA[1674,12] := 2.21055;
   DATA[1674,13] := 866.084;
   DATA[1674,14] := 1.0;
   DATA[1674,15] := 2.0;
   DATA[1674,16] := 1.0;
   DATA[1674,17] := 1.0;
   DATA[1674,18] := 1.0;
   DATA[1674,19] := 2.0;
   DATA[1674,20] := 148.808;
   DATA[1674,21] := 153.9862;
   DATA[1674,22] := 1.713261;
   DATA[1674,23] := 801.1023;
   DATA[1674,24] := 2.0;
   DATA[1674,25] := 2.0;
   DATA[1674,26] := 7.876058;
   DATA[1674,27] := 142.9377;
   DATA[1674,28] := 262.6891;
   DATA[1674,29] := 12.15073;
   DATA[1674,30] := 1.721866;
   DATA[1674,31] := 1.271679;
   DATA[1674,32] := 0.7355248;
   DATA[1674,33] := 0.3082983;
   DATA[1674,34] := 2.0;
   DATA[1674,35] := 249.7597;
   DATA[1674,36] := 1.585878;
   DATA[1674,37] := 188.7337;
   DATA[1674,38] := 0.000128152;
   DATA[1674,39] := 1.0;
   DATA[1675,1] := 815.5153;
   DATA[1675,2] := 1.0;
